Yaskawa INFORM job: SKRZYNIA_4040_180_STOPNI_10B_NEW.JBI

/JOB
//NAME SKRZYNIA_4040_180_STOPNI_10B_NEW
///FOLDERNAME 02-SKRZYNIE_JOBS
//POS
///NPOS 723,723,0,26,0,0
///TOOL 0
///POSTYPE PULSE
///PULSE
C00000=-21231,-51303,42314,2367,6591,-1439
C00001=-12854,-61498,-6635,149088,-29435,16513
C00002=84284,-61498,-6635,149088,14842,16513
C00003=84426,-61498,-62039,149088,14842,16513
C00004=84426,-61498,-83719,149088,14842,16513
C00005=40079,-25830,-61904,72398,37828,17494
C00006=40079,-25830,-61904,72398,37828,17494
C00007=38824,-23395,-60038,72349,38727,17731
C00008=41545,-22667,-59464,70826,37145,18191
C00009=40079,-25830,-61904,72398,37828,17494
C00010=40079,-23879,-31232,97616,36989,2612
C00011=40241,-22903,-30855,97033,36795,2952
C00012=39596,-21803,-29985,96678,37187,3182
C00013=41542,-21522,-29763,96797,35874,3054
C00014=40241,-22903,-30855,97033,36795,2952
C00015=44500,-22967,-34027,49689,40772,15208
C00016=44759,-21950,-33222,49364,40770,15399
C00017=43898,-20603,-32137,49608,41392,15289
C00018=45676,-20288,-31878,48567,40497,15854
C00019=44759,-21950,-33222,49364,40770,15399
C00020=50639,-31838,-53853,40430,42590,20636
C00021=47737,-42531,-47731,84740,46626,-3202
C00022=73324,-51450,-15857,136644,48513,-27329
C00023=28578,-31257,-33285,101874,54895,-3139
C00024=29101,-23166,-41439,93785,52323,3372
C00025=30342,-16402,-40775,90158,51109,6027
C00026=29555,-14242,-38855,90054,51607,6222
C00027=31304,-14182,-38798,89754,50458,6198
C00028=30342,-16402,-40775,90158,51109,6027
C00029=37840,-26567,-47806,97824,39338,5403
C00030=38314,-22656,-45541,96192,38787,6352
C00031=38740,-21749,-44817,95954,38481,6451
C00032=38106,-20505,-43805,95701,38856,6673
C00033=39920,-20274,-43616,95549,37666,6573
C00034=38740,-21749,-44817,95954,38481,6451
C00035=35154,-23288,-28184,89821,43405,2441
C00036=35403,-21021,-26397,89340,43215,2751
C00037=34678,-19569,-25213,89063,43699,2948
C00038=36545,-19419,-25091,89018,42427,2940
C00039=35403,-21021,-26397,89340,43215,2751
C00040=46673,-28267,-59493,36306,49500,22578
C00041=47298,-25083,-54483,36432,48421,22382
C00042=46134,-23276,-53085,36983,49197,22170
C00043=48093,-22778,-52692,35651,48513,22818
C00044=47298,-25083,-54483,36432,48421,22382
C00045=72417,-67880,-88171,46465,42262,31903
C00046=81480,-74508,-67932,111005,17511,3722
C00047=42492,-36415,-29790,92406,42740,11684
C00048=46673,-28267,-59493,36306,49500,22578
C00049=47298,-25083,-54483,36432,48421,22382
C00050=46134,-23276,-53085,36983,49197,22170
C00051=48093,-22778,-52692,35651,48513,22818
C00052=47298,-25083,-54483,36432,48421,22382
C00053=46673,-28267,-59493,36306,49500,22578
C00054=47298,-25083,-54483,36432,48421,22382
C00055=46134,-23276,-53085,36983,49197,22170
C00056=48093,-22778,-52692,35651,48513,22818
C00057=47309,-25052,-54460,36421,48423,22388
C00058=43000,-32780,-49011,53703,41088,15214
C00059=66148,-65994,-55487,105361,28212,-7739
C00060=66148,-65994,-55487,105361,28212,-7739
C00061=59848,-54778,-49507,133915,29212,-10807
C00062=45497,-38347,-41839,114412,32622,-465
C00063=46376,-32635,-46933,102993,29107,5780
C00064=46303,-28031,-46898,97061,28371,8976
C00065=45038,-26161,-45521,96183,29128,9541
C00066=46946,-25787,-45238,96120,27855,9431
C00067=46303,-28031,-46898,97061,28371,8976
C00068=45864,-17128,1685,129467,40696,-9274
C00069=46023,-15894,1830,128891,40053,-8896
C00070=45181,-14790,2774,128176,40341,-8535
C00071=46921,-14545,2986,129317,39465,-9073
C00072=45402,-17127,796,128656,40504,-8810
C00073=42828,-21985,-11573,106778,34538,-1929
C00074=43349,-21404,-11124,106831,34165,-1930
C00075=42250,-19876,-9917,105946,34757,-1485
C00076=44494,-19460,-9583,106781,33302,-1837
C00077=42797,-21858,-11474,106726,34550,-1903
C00078=42956,-14057,7354,88292,32197,-569
C00079=43438,-13569,7781,88275,31880,-510
C00080=42549,-12302,8904,87823,32462,-349
C00081=44721,-11883,9282,88161,31033,-316
C00082=42944,-14884,6642,88491,32210,-682
C00083=72417,-67880,-88171,46465,42262,31903
C00084=81480,-74508,-67932,111005,17511,3722
C00085=42492,-36415,-29790,92406,42740,11684
C00086=29699,-14901,-14062,86637,51249,15251
C00087=28921,-12904,-12269,86425,51786,15406
C00088=30978,-12767,-12144,86426,50380,15429
C00089=29506,-17416,-16239,86937,51377,15018
C00090=88410,-69609,-60867,139529,19008,-8209
C00091=62412,-62489,-12046,-12266,17816,34850
C00092=7585,-53665,33325,-3309,7810,4157
C00093=-681,-52632,38645,-5695,5489,-631
C00094=-17840,-61498,-6635,-149088,-29435,-16513
C00095=-84284,-61498,-6635,-149088,14842,-16513
C00096=-84426,-61498,-62039,-149088,14842,-16513
C00097=-84426,-61498,-83719,-149088,14842,-16513
C00098=-83351,-27062,-60322,-167360,37385,6517
C00099=-83351,-27062,-60322,-167360,37385,23281
C00100=-45097,-23850,-79932,-76262,26943,-22849
C00101=-48253,-15729,-73342,-71138,25693,-24842
C00102=-50302,-13076,-73239,-65836,25323,-27140
C00103=-49401,-11675,-71961,-66260,25816,-27133
C00104=-50608,-11574,-71867,-65226,25249,-27391
C00105=-49660,-13361,-73494,-66442,25615,-26975
C00106=-48242,-21102,-77802,-73044,25430,-23851
C00107=-42432,-29691,-46140,-101591,34194,-3953
C00108=-40467,-32259,-45349,-89481,35752,-6083
C00109=-35590,-22323,-38089,-87474,43148,-7978
C00110=-34853,-20780,-36847,-87247,43643,-8181
C00111=-37029,-20471,-36594,-86926,42180,-8224
C00112=-35503,-23333,-38886,-87700,43207,-7835
C00113=-41659,-25848,-37197,-61468,39541,-12344
C00114=-42019,-23363,-32043,-63110,38591,-11327
C00115=-41283,-22167,-31102,-63128,39154,-11341
C00116=-43189,-21868,-30866,-62281,38009,-11788
C00117=-40846,-25460,-35158,-62968,39555,-11455
C00118=-39561,-32409,-42051,-71473,38885,-9254
C00119=-88477,-67032,-53890,-125185,13082,17955
C00120=-90715,-66667,-50935,-152816,24533,28486
C00121=-30735,-26920,-32844,-95116,50209,-1071
C00122=-37180,-24683,-31930,-114741,47007,2943
C00123=-36407,-19634,-34656,-109847,45004,-453
C00124=-38352,-16604,-33863,-108521,43129,-1176
C00125=-37479,-14809,-32279,-108169,43576,-1482
C00126=-39395,-14487,-31992,-108361,42368,-1194
C00127=-37253,-18321,-35339,-108644,43916,-1187
C00128=-30948,-19486,-27368,-89515,49970,-2899
C00129=-32453,-17458,-25663,-89179,48933,-3088
C00130=-31896,-16151,-24534,-89028,49305,-3221
C00131=-33527,-16125,-24510,-88960,48196,-3202
C00132=-31291,-18911,-26892,-89421,49733,-2955
C00133=-32789,-14788,-10714,-75998,48642,-1904
C00134=-33953,-13481,-9550,-75758,47902,-2112
C00135=-33380,-12226,-8408,-75670,48319,-2157
C00136=-35020,-12164,-8351,-75529,47228,-2306
C00137=-33300,-14767,-10697,-75957,48300,-1949
C00138=-33300,-14767,-10697,-75957,48300,-1949
C00139=-33901,-13199,-7224,-76945,47663,-1266
C00140=-33178,-11617,-5779,-76815,48184,-1329
C00141=-35129,-11426,-5603,-76688,46886,-1497
C00142=-32900,-14718,-9841,-76444,48459,-1584
C00143=-74406,-60637,-53290,-78600,32734,-4861
C00144=-66351,-49775,-22313,-121187,42752,19491
C00145=-38126,-18978,-6321,-103556,42156,4232
C00146=-33300,-14767,-10697,-75957,48300,-1949
C00147=-33901,-13199,-7224,-76945,47663,-1266
C00148=-33178,-11617,-5779,-76815,48184,-1329
C00149=-35129,-11426,-5603,-76688,46886,-1497
C00150=-32900,-14718,-9841,-76444,48459,-1584
C00151=-33300,-14767,-10697,-75957,48300,-1949
C00152=-33901,-13199,-7224,-76945,47663,-1266
C00153=-33178,-11617,-5779,-76815,48184,-1329
C00154=-35129,-11426,-5603,-76688,46886,-1497
C00155=-33596,-13726,-8578,-76506,47971,-1566
C00156=-46324,-38325,-53351,-48650,39022,-16558
C00157=-84678,-53272,-42524,-56273,5220,-14251
C00158=-79949,-57830,-54545,-43165,18800,-25262
C00159=-85199,-63426,-59279,-35356,8253,-25340
C00160=-43240,-40066,-69296,-76804,34492,-13950
C00161=-32352,-24302,-62495,-76398,48702,-17646
C00162=-33867,-19497,-59989,-74208,48202,-18898
C00163=-33043,-17469,-58279,-74274,48770,-19034
C00164=-35172,-17180,-58031,-73305,47532,-19251
C00165=-33150,-20833,-61090,-74721,48572,-18687
C00166=-32525,-19963,-22291,-97454,48417,-2656
C00167=-34479,-17146,-19937,-97221,47013,-2812
C00168=-33716,-15515,-18525,-96928,47480,-3025
C00169=-35357,-15455,-18472,-97073,46375,-2908
C00170=-33341,-18474,-21063,-97306,47817,-2759
C00171=-32838,-10388,7981,-94473,48357,2926
C00172=-33747,-9461,8037,-94117,47673,2571
C00173=-33094,-8062,9377,-93861,48090,2458
C00174=-34952,-7927,9507,-94260,46861,2543
C00175=-33010,-10379,7174,-94037,48174,2591
C00176=-36099,-20774,-22249,-70758,44565,-7624
C00177=-37926,-16067,-12890,-73276,42575,-5996
C00178=-37323,-14944,-11908,-73188,43017,-6038
C00179=-39053,-14785,-11769,-72915,41882,-6255
C00180=-37847,-19214,-17221,-72670,42783,-6386
C00181=-74406,-60637,-53290,-78600,32734,-4861
C00182=-66351,-49775,-22313,-121187,42752,19491
C00183=-38126,-18978,-6321,-103556,42156,4232
C00184=-39485,-17529,-8330,-90200,39091,223
C00185=-38315,-15563,-6658,-89669,39866,-39
C00186=-40130,-15376,-6497,-89855,38637,-21
C00187=-40610,-23081,-12745,-91737,38407,1092
C00188=-82794,-45547,-18103,-153793,26453,27163
C00189=-46099,-67236,-11725,-98004,28606,19827
C00190=275,-40498,62911,330,272,-175
C00191=-21231,-51303,42314,2367,6591,-1439
C00192=-12854,-61498,-6635,149088,-29435,16513
C00193=84284,-61498,-6635,149088,14842,16513
C00194=84426,-61498,-62039,149088,14842,16513
C00195=84426,-61498,-83719,149088,14842,16513
C00196=40079,-25830,-61904,72398,37828,17494
C00197=43542,-21744,-53414,85694,32141,12908
C00198=43538,-20959,-59091,78847,32551,16732
C00199=40079,-23879,-31232,97616,36989,2612
C00200=41069,-22296,-36683,87871,35939,7163
C00201=41069,-20857,-27994,94343,36275,3375
C00202=40241,-22903,-30855,97033,36795,2952
C00203=44500,-22967,-34027,49689,40772,15208
C00204=37674,-14410,-29425,54908,51799,12689
C00205=37617,-13106,-20810,58248,49229,10178
C00206=44759,-21950,-33222,49364,40770,15399
C00207=50639,-31838,-53853,40430,42590,20636
C00208=47737,-42531,-47731,84740,46626,-3202
C00209=78714,-49092,-28755,133609,38199,-24420
C00210=28578,-31257,-33285,101874,54895,-3139
C00211=29101,-23166,-41439,93785,52323,3372
C00212=31163,-13872,-34138,92103,50752,4440
C00213=31163,-14064,-41434,88282,50498,7326
C00214=30342,-16402,-40775,90158,51109,6027
C00215=37840,-26567,-47806,97824,39338,5403
C00216=38314,-22656,-45541,96192,38787,6352
C00217=39658,-19881,-39017,99036,38353,4498
C00218=39658,-20227,-46296,93241,37598,7980
C00219=38740,-21749,-44817,95954,38481,6451
C00220=35154,-23288,-28184,89821,43405,2441
C00221=36302,-20456,-32356,81251,42995,6506
C00222=36302,-19046,-24537,85721,42698,3608
C00223=35403,-21021,-26397,89340,43215,2751
C00224=46673,-28267,-59493,36306,49500,22578
C00225=35383,-14910,-45807,52457,59655,19882
C00226=35383,-15025,-38926,54776,56903,17744
C00227=47298,-25083,-54483,36432,48421,22382
C00228=72417,-64226,-72669,53660,37323,27470
C00229=81480,-74508,-67932,111005,17511,3722
C00230=31559,-23192,-27729,97069,50041,14774
C00231=31559,-23192,-27729,97069,50041,14774
C00232=46673,-28267,-59493,36306,49500,22578
C00233=37754,-20085,-42350,56977,49558,11229
C00234=37583,-19171,-35264,59813,47966,9525
C00235=50836,-29533,-47785,41620,34114,14584
C00236=46673,-28267,-59493,36306,49500,22578
C00237=35383,-14910,-45807,52457,59655,19882
C00238=35383,-15025,-38926,54776,56903,17744
C00239=40792,-20879,-47843,46282,52305,19657
C00240=43000,-32780,-49011,53703,41088,15214
C00241=90538,-65158,-52413,145953,6697,-22013
C00242=90538,-65158,-52413,145953,6697,-22013
C00243=59848,-54778,-49507,133915,29212,-10807
C00244=45497,-38347,-41839,114412,32622,-465
C00245=46376,-32635,-46933,102993,29107,5780
C00246=38443,-20223,-37840,96971,39567,10287
C00247=38443,-20698,-44956,91660,38993,13539
C00248=46303,-28031,-46898,97061,28371,8976
C00249=45864,-17128,1685,129467,40696,-9274
C00250=38069,-7942,12691,120284,49952,-5070
C00251=38069,-11604,1369,116685,47266,-2469
C00252=45402,-17127,796,128656,40504,-8810
C00253=42828,-21985,-11573,106778,34538,-1929
C00254=33281,-15275,-13406,92642,47209,4970
C00255=33281,-12456,-2996,97026,47894,1870
C00256=42797,-21858,-11474,106726,34550,-1903
C00257=42956,-14057,7354,88292,32197,-569
C00258=35915,-8349,8335,81338,43542,2014
C00259=35915,-4149,20758,86814,43229,-1568
C00260=42944,-14884,6642,88491,32210,-682
C00261=72417,-64226,-72669,53660,37323,27470
C00262=81480,-74508,-67932,111005,17511,3722
C00263=31559,-23192,-27729,97069,50041,14774
C00264=31559,-23192,-27729,97069,50041,14774
C00265=34921,-13948,-26935,108215,46513,15013
C00266=34921,-14719,-34056,104413,45059,17611
C00267=30729,-14807,-22031,91030,50318,16982
C00268=30729,-14807,-22031,91030,50318,16982
C00269=30729,-13019,-13516,94566,50766,14318
C00270=88410,-69609,-60867,139529,19008,-8209
C00271=62412,-62489,-12046,-12266,17816,34850
C00272=-245,-52407,39795,-2053,6376,-227
C00273=-681,-52632,38645,-5695,5489,-631
C00274=-17840,-61498,-6635,-149088,-29435,-16513
C00275=-84284,-61498,-6635,-149088,14842,-16513
C00276=-84426,-61498,-62039,-149088,14842,-16513
C00277=-84426,-61498,-83719,-149088,14842,-16513
C00278=-83351,-27062,-60322,-167360,37385,6517
C00279=-83351,-27062,-60322,-167360,37385,23281
C00280=-45097,-23850,-79932,-76262,26943,-22849
C00281=-48253,-15729,-73342,-71138,25693,-24842
C00282=-42869,-6204,-67496,-75794,33821,-25861
C00283=-42869,-3205,-70686,-69723,34977,-29338
C00284=-49660,-13361,-73494,-66442,25615,-26975
C00285=-48242,-21102,-77802,-73044,25430,-23851
C00286=-42432,-29691,-46140,-101591,34194,-3953
C00287=-40467,-32259,-45349,-89481,35752,-6083
C00288=-32032,-15700,-34761,-86363,49905,-9645
C00289=-32032,-14866,-27372,-89947,49973,-6979
C00290=-35503,-23333,-38886,-87700,43207,-7835
C00291=-41659,-25848,-37197,-61468,39541,-12344
C00292=-32550,-13183,-23016,-68651,53358,-8526
C00293=-34023,-12481,-22084,-63241,53452,-9524
C00294=-40846,-25460,-35158,-62968,39555,-11455
C00295=-39561,-32409,-42051,-71473,38885,-9254
C00296=-88477,-67032,-53890,-125185,13082,17955
C00297=-90715,-66667,-50935,-152816,24533,28486
C00298=-30735,-26920,-32844,-95116,50209,-1071
C00299=-37180,-24683,-31930,-114741,47007,2943
C00300=-36407,-19634,-34656,-109847,45004,-453
C00301=-39264,-14095,-28560,-110319,43249,69
C00302=-39254,-14742,-35710,-105973,41627,-2729
C00303=-37253,-18321,-35339,-108644,43916,-1187
C00304=-30948,-19486,-27368,-89515,49970,-2899
C00305=-33188,-17217,-33290,-80523,49125,-7157
C00306=-33231,-16133,-25752,-84153,48705,-4513
C00307=-31291,-18911,-26892,-89421,49733,-2955
C00308=-32789,-14788,-10714,-75998,48642,-1904
C00309=-32456,-10000,-8763,-74569,51725,-2878
C00310=-32456,-7502,814,-78111,50801,-165
C00311=-33300,-14767,-10697,-75957,48300,-1949
C00312=-33300,-14767,-10697,-75957,48300,-1949
C00313=-31039,-7597,-4415,-75714,54029,-1891
C00314=-31745,-5891,1281,-74609,53027,-1007
C00315=-32900,-14718,-9841,-76444,48459,-1584
C00316=-73757,-59015,-49060,-81128,30370,-3444
C00317=-66351,-49775,-22313,-115582,40632,19491
C00318=-39230,-13378,9505,-118180,46878,7841
C00319=-33300,-14767,-10697,-75957,48300,-1949
C00320=-31039,-7597,-4415,-75714,54029,-1891
C00321=-31745,-5891,1281,-74609,53027,-1007
C00322=-32900,-14718,-9841,-76444,48459,-1584
C00323=-33300,-14767,-10697,-75957,48300,-1949
C00324=-31039,-7597,-4415,-75714,54029,-1891
C00325=-31745,-5891,1281,-74609,53027,-1007
C00326=-31800,-10328,-6603,-75899,51910,-1826
C00327=-46324,-38325,-53351,-48650,39022,-16558
C00328=-84678,-53272,-42524,-56273,5220,-14251
C00329=-79949,-57830,-54545,-43165,18800,-25262
C00330=-85199,-63426,-59279,-35356,8253,-25340
C00331=-43240,-40066,-69296,-76804,34492,-13950
C00332=-32352,-24302,-62495,-76398,48702,-17646
C00333=-34311,-15084,-43386,-89458,46770,-12174
C00334=-34303,-14562,-49859,-85086,46777,-15220
C00335=-33150,-20833,-61090,-74721,48572,-18687
C00336=-32525,-19963,-22291,-97454,48417,-2656
C00337=-35706,-13608,-12356,-102024,46946,-662
C00338=-35706,-15621,-21438,-97808,45877,-3577
C00339=-33341,-18474,-21063,-97306,47817,-2759
C00340=-32838,-10388,7981,-94473,48357,2926
C00341=-33093,-7396,5806,-90907,49596,566
C00342=-33114,-3922,16616,-94789,50065,3444
C00343=-33010,-10379,7174,-94037,48174,2591
C00344=-36099,-20774,-22249,-70758,44565,-7624
C00345=-34715,-11750,-12273,-72011,49148,-6727
C00346=-34715,-9605,-3694,-75523,48112,-4187
C00347=-37847,-19214,-17221,-72670,42783,-6386
C00348=-73757,-59015,-49060,-81128,30370,-3444
C00349=-66351,-49775,-22313,-115582,40632,19491
C00350=-39230,-13378,9505,-118180,46878,7841
C00351=-45382,-7236,12023,-133378,48537,9962
C00352=-45404,-10871,608,-130166,44845,7725
C00353=-39289,-13633,5656,-114159,44810,6160
C00354=-38323,-13232,3563,-106275,42852,3854
C00355=-39624,-12309,2722,-105485,41613,3229
C00356=-39624,-8328,14658,-110578,43519,6514
C00357=-36264,-16485,7382,-110054,45980,6615
C00358=-44249,-32643,-4456,-118298,43922,12613
C00359=-31781,-48654,10305,-108801,40875,18482
C00360=275,-40498,62911,330,272,-175
C00361=-21231,-51303,42314,2367,6591,-1439
C00362=-12854,-61498,-6635,149088,-29435,16513
C00363=1243,-64916,-20173,127712,-3737,19309
C00364=25728,-72945,-47671,86292,40512,26238
C00365=76664,-93599,-96338,114349,24908,7990
C00366=72545,-76403,-90681,98079,12187,16258
C00367=68435,-42241,-79282,43384,21203,43145
C00368=65057,-16377,-54230,51764,24572,24912
C00369=65057,-16377,-54230,51764,24572,24912
C00370=63338,-14509,-52578,53100,25585,24479
C00371=65493,-13068,-51269,50530,24633,25485
C00372=65057,-16377,-54230,51764,24572,24912
C00373=65057,-15356,-24189,99795,20011,765
C00374=64877,-14372,-23690,98704,20045,1316
C00375=64002,-13489,-22890,98156,20604,1621
C00376=65592,-12702,-22173,98357,19527,1466
C00377=64877,-14372,-23690,98704,20045,1316
C00378=68341,-13254,-25781,29903,31229,25524
C00379=68283,-12212,-24821,29865,31356,25548
C00380=67188,-11145,-23825,30867,31841,25051
C00381=68624,-10377,-23095,29361,31405,25809
C00382=68283,-12212,-24821,29865,31356,25548
C00383=67373,-28813,-51747,26561,36937,27500
C00384=65665,-56911,-59086,75825,31170,1181
C00385=86238,-56758,-47218,93606,16664,-7096
C00386=86238,-56758,-47218,93606,16664,-7096
C00387=58162,-25487,-29222,106212,35121,-6052
C00388=54729,-17550,-36821,90686,35172,3055
C00389=53879,-10723,-35593,84994,35691,6442
C00390=52628,-8898,-33837,85063,36512,6546
C00391=54193,-8333,-33282,84633,35489,6620
C00392=53879,-10723,-35593,84994,35691,6442
C00393=63265,-18185,-41125,95483,22448,4389
C00394=62561,-14368,-38517,92984,22773,5727
C00395=62689,-13396,-37636,92694,22678,5861
C00396=61812,-12400,-36718,92465,23238,6064
C00397=63331,-11679,-36046,92201,22238,6052
C00398=62689,-13396,-37636,92694,22678,5861
C00399=60836,-16142,-22303,87853,25853,3109
C00400=60346,-13901,-20318,87240,26185,3441
C00401=59279,-12702,-19226,86999,26911,3593
C00402=60868,-12050,-18626,86765,25831,3679
C00403=60346,-13901,-20318,87240,26185,3441
C00404=71174,-16943,-50501,16787,44328,31924
C00405=70846,-13961,-45205,17496,43056,31510
C00406=69412,-12602,-43961,18675,43507,30969
C00407=70949,-11616,-43043,17320,43301,31610
C00408=70846,-13961,-45205,17496,43056,31510
C00409=75423,-38775,-29488,68062,11357,11878
C00410=83800,-53438,-37305,103753,25026,-1265
C00411=73693,-43023,-29306,101200,31062,8332
C00412=71174,-16943,-50501,16787,44328,31924
C00413=70846,-13961,-45205,17496,43056,31510
C00414=69412,-12602,-43961,18675,43507,30969
C00415=70949,-11616,-43043,17320,43301,31610
C00416=70846,-13961,-45205,17496,43056,31510
C00417=71174,-16943,-50501,16787,44328,31924
C00418=70846,-13961,-45205,17496,43056,31510
C00419=69412,-12602,-43961,18675,43507,30969
C00420=70949,-11616,-43043,17320,43301,31610
C00421=70341,-14112,-45346,17938,43139,31306
C00422=66765,-25643,-43957,33958,30926,25005
C00423=89904,-51519,-74342,14421,36812,44678
C00424=59533,-60921,-66479,83565,41795,11392
C00425=74572,-27669,-34920,136415,14797,-11887
C00426=72479,-21736,-38943,108586,11547,1590
C00427=70901,-17325,-38411,94105,11830,8638
C00428=69318,-15905,-37172,92885,12849,9347
C00429=70820,-15051,-36412,92531,11846,9399
C00430=70901,-17325,-38411,94105,11830,8638
C00431=70927,-7523,10343,151197,29871,-19432
C00432=70517,-6236,10737,150221,29352,-18933
C00433=69462,-5331,11645,148944,29606,-18324
C00434=70849,-4645,12343,150548,29173,-19084
C00435=70402,-7634,9356,150158,29478,-18907
C00436=68660,-13051,-4106,122816,18275,-8999
C00437=68895,-12351,-3471,122899,18094,-9031
C00438=67458,-11121,-2337,120787,18802,-8043
C00439=69212,-10147,-1425,122703,17774,-8922
C00440=68590,-12934,-4000,122687,18305,-8939
C00441=67960,-5141,15741,92957,15720,-628
C00442=68207,-4523,16370,92944,15555,-601
C00443=67051,-3465,17460,92338,16311,-404
C00444=68762,-2475,18496,92897,15183,-531
C00445=68227,-5981,14898,93242,15553,-745
C00446=75423,-38775,-29488,68062,11357,11878
C00447=83800,-53438,-37305,103753,25026,-1265
C00448=73693,-43023,-29306,101200,31062,8332
C00449=57182,-8361,13896,122065,42938,1264
C00450=54175,-4244,10116,111777,38351,4895
C00451=53015,-2664,11762,111180,39035,5172
C00452=54334,-2350,12093,111780,38228,4906
C00453=54175,-4244,10116,111777,38351,4895
C00454=89016,-59505,-36896,143842,20811,-11822
C00455=0,-52280,40443,0,6876,0
C00456=-681,-52632,38645,-5695,5489,-631
C00457=-17840,-61498,-6635,-149088,-29435,-16513
C00458=-84284,-61498,-6635,-149088,14842,-16513
C00459=-57949,-92832,-68327,-119114,39180,-13331
C00460=-51160,-78996,-68705,-103851,38676,-21739
C00461=-70129,-12201,-70194,-45988,15849,-32683
C00462=-70861,-4247,-62448,-43170,16032,-33903
C00463=-72229,-1292,-61598,-37253,16795,-36501
C00464=-71164,-286,-60510,-39045,17142,-35862
C00465=-72168,114,-60071,-37345,16819,-36474
C00466=-71747,-1710,-62044,-38091,16943,-36199
C00467=-72086,-8949,-67137,-41785,15362,-34318
C00468=-68226,-19972,-38714,-103620,16923,-1218
C00469=-67549,-22986,-38612,-80975,17520,-9124
C00470=-60286,-14955,-31870,-81576,26630,-9634
C00471=-59206,-13694,-30736,-81541,27366,-9725
C00472=-61026,-12796,-29913,-80837,26167,-9971
C00473=-60502,-15936,-32740,-81790,26471,-9505
C00474=-66711,-16726,-29834,-42060,26790,-21996
C00475=-66477,-14329,-24475,-44917,25565,-20507
C00476=-65503,-13376,-23611,-45716,26132,-20127
C00477=-67048,-12587,-22889,-44009,25442,-20959
C00478=-66009,-16611,-27996,-44380,26285,-20808
C00479=-67084,-23473,-35621,-52822,22843,-18344
C00480=-54372,-63877,-56403,-90862,27079,1323
C00481=-55608,-75012,-34654,-126966,55573,20814
C00482=-55608,-75012,-34654,-126966,55573,20814
C00483=-58069,-20780,-28125,-95622,31565,-134
C00484=-62818,-16895,-25617,-123146,31403,8811
C00485=-60301,-12189,-28106,-114654,29999,4030
C00486=-61167,-8731,-26593,-112607,28768,2985
C00487=-59960,-7252,-25135,-111997,29446,2563
C00488=-61574,-6413,-24296,-112502,28453,2957
C00489=-60636,-10677,-28466,-112685,29164,2987
C00490=-55814,-13636,-22293,-87541,33030,-3263
C00491=-56566,-11270,-20110,-87077,32519,-3496
C00492=-55709,-10167,-19066,-86969,33101,-3589
C00493=-57154,-9687,-18605,-86794,32120,-3632
C00494=-55949,-12989,-21706,-87412,32939,-3330
C00495=-57109,-8613,-4995,-71756,32687,-5152
C00496=-57764,-7017,-3429,-71410,32292,-5358
C00497=-56909,-5946,-2356,-71529,32873,-5273
C00498=-58347,-5433,-1836,-71115,31941,-5534
C00499=-57555,-8453,-4841,-71622,32398,-5235
C00500=-57555,-8453,-4841,-71622,32398,-5235
C00501=-57844,-6749,-1100,-73475,31868,-4209
C00502=-56760,-5394,262,-73573,32605,-4123
C00503=-58439,-4668,1002,-73167,31507,-4396
C00504=-57269,-8513,-4090,-72514,32435,-4729
C00505=-69972,-70945,-58827,-87515,35615,-17
C00506=-69972,-70945,-58827,-87515,35615,-17
C00507=-64053,-11295,342,-114563,25508,8776
C00508=-57555,-8453,-4841,-71622,32398,-5235
C00509=-57844,-6749,-1100,-73475,31868,-4209
C00510=-56760,-5394,262,-73573,32605,-4123
C00511=-58439,-4668,1002,-73167,31507,-4396
C00512=-57269,-8513,-4090,-72514,32435,-4729
C00513=-57555,-8453,-4841,-71622,32398,-5235
C00514=-57844,-6749,-1100,-73475,31868,-4209
C00515=-56760,-5394,262,-73573,32605,-4123
C00516=-58439,-4668,1002,-73167,31507,-4396
C00517=-57340,-8164,-3656,-72551,32379,-4710
C00518=-74194,-26905,-45748,-21164,30431,-30370
C00519=-93036,-61583,-83098,-4972,39040,-38907
C00520=-93036,-61583,-83098,-4972,39040,-38907
C00521=-71878,-28414,-61729,-48672,19032,-25171
C00522=-58025,-17185,-56692,-61796,34178,-22014
C00523=-58138,-12270,-53641,-59720,34855,-23185
C00524=-56898,-10637,-52111,-60384,35596,-23031
C00525=-58712,-9745,-51261,-58987,34681,-23500
C00526=-57851,-13714,-54968,-60141,34926,-22995
C00527=-57767,-13689,-16896,-100181,31334,-836
C00528=-58645,-10437,-13885,-99794,30663,-1040
C00529=-57513,-9065,-12573,-99347,31388,-1300
C00530=-58947,-8556,-12078,-99591,30423,-1148
C00531=-58031,-12031,-15383,-99926,31110,-974
C00532=-57646,-4162,14084,-101426,32077,4804
C00533=-58050,-2999,14481,-100683,31666,4357
C00534=-57067,-1784,15765,-100255,32298,4198
C00535=-58672,-1130,16464,-100866,31256,4407
C00536=-57676,-4116,13320,-100600,31921,4338
C00537=-61201,-13510,-16039,-60848,29053,-13371
C00538=-61885,-8475,-5914,-65722,27292,-10768
C00539=-61040,-7537,-4993,-65975,27855,-10622
C00540=-62506,-6917,-4380,-65230,26947,-11038
C00541=-62587,-11561,-10517,-63923,27184,-11731
C00542=-69972,-70945,-58827,-87515,35615,-17
C00543=-69972,-70945,-58827,-87515,35615,-17
C00544=-64053,-11295,342,-114563,25508,8776
C00545=-64305,-9514,-1154,-92513,22236,350
C00546=-62690,-7882,422,-91839,23314,70
C00547=-64201,-7220,1072,-92034,22288,112
C00548=-67149,-14673,-5883,-94845,20391,1413
C00549=-66017,-67071,-29713,-134523,32873,22112
C00550=-46099,-67236,-11725,-98004,28606,19827
C00551=275,-40498,62911,330,272,-175
C00552=-21231,-51303,42314,2367,6591,-1439
C00553=-12854,-61498,-6635,149088,-29435,16513
C00554=84284,-61498,-6635,149088,14842,16513
C00555=84426,-61498,-62039,149088,14842,16513
C00556=84426,-61498,-83719,149088,14842,16513
C00557=65057,-16377,-54230,51764,24572,24912
C00558=84197,-12836,-45810,-45141,8815,68584
C00559=84197,-12041,-51210,-30828,12194,61758
C00560=65057,-15356,-24189,99795,20011,765
C00561=74080,-15423,-30907,69143,7686,14038
C00562=74080,-14352,-23480,100923,7503,-991
C00563=64877,-14372,-23690,98704,20045,1316
C00564=68341,-13254,-25781,29903,31229,25524
C00565=74439,-11496,-26749,13621,29642,33649
C00566=74439,-10401,-19085,15788,25340,32499
C00567=68283,-12212,-24821,29865,31356,25548
C00568=75452,-19560,-44582,17787,36745,31835
C00569=68183,-44834,-62310,40554,34116,19994
C00570=94103,-63119,-69903,16230,17694,31762
C00571=91219,-55958,-51219,93435,14423,-1742
C00572=58162,-25487,-29222,106212,35121,-6052
C00573=54729,-17550,-36821,90686,35172,3055
C00574=70769,-15160,-35297,83470,11760,4000
C00575=70769,-15377,-40609,67973,12489,11436
C00576=53879,-10723,-35593,84994,35691,6442
C00577=63265,-18185,-41125,95483,22448,4389
C00578=62561,-14368,-38517,92984,22773,5727
C00579=77715,-13962,-33882,144680,4496,-21400
C00580=77806,-14046,-41277,60589,2532,18064
C00581=62689,-13396,-37636,92694,22678,5861
C00582=60836,-16142,-22303,87853,25853,3109
C00583=74678,-16514,-29029,42946,9451,23276
C00584=74678,-15315,-21920,65026,7151,12815
C00585=60346,-13901,-20318,87240,26185,3441
C00586=71174,-16943,-50501,16787,44328,31924
C00587=80494,-13102,-44599,-1731,38384,44653
C00588=80494,-13295,-38861,-1907,34285,44756
C00589=70846,-13961,-45205,17496,43056,31510
C00590=83595,-66668,-34414,154325,14846,-28455
C00591=83595,-66668,-34414,154325,14846,-28455
C00592=69137,-30288,-25983,94330,24536,11676
C00593=71174,-16943,-50501,16787,44328,31924
C00594=80494,-13102,-44599,-1731,38384,44653
C00595=80494,-13295,-38861,-1907,34285,44756
C00596=70846,-13961,-45205,17496,43056,31510
C00597=71056,-15939,-48723,17027,43904,31784
C00598=80494,-13102,-44599,-1731,38384,44653
C00599=80494,-13295,-38861,-1907,34285,44756
C00600=73484,-14077,-43720,13005,40199,34803
C00601=69645,-22678,-41665,30358,30421,26767
C00602=81017,-78801,-66317,80675,7786,2447
C00603=81017,-78801,-66317,80675,7786,2447
C00604=74572,-27669,-34920,136415,14797,-11887
C00605=72479,-21736,-38943,108586,11547,1590
C00606=76162,-15538,-34076,119407,5153,-4143
C00607=76225,-15803,-40874,66675,4586,20654
C00608=70901,-17325,-38411,94105,11830,8638
C00609=70927,-7523,10343,151197,29871,-19432
C00610=75273,-951,23395,164730,33684,-27271
C00611=75257,-4812,11918,163197,28775,-26429
C00612=70402,-7634,9356,150158,29478,-18907
C00613=68660,-13051,-4106,122816,18275,-8999
C00614=75422,-13779,-12311,124767,7049,-10125
C00615=75402,-11409,-3274,143452,10422,-18986
C00616=68590,-12934,-4000,122687,18305,-8939
C00617=67960,-5141,15741,92957,15720,-628
C00618=77005,-5383,11265,73049,3770,10304
C00619=77005,-1367,23224,135174,5603,-18901
C00620=68227,-5981,14898,93242,15553,-745
C00621=83595,-66668,-34414,154325,14846,-28455
C00622=83595,-66668,-34414,154325,14846,-28455
C00623=69137,-30288,-25983,94330,24536,11676
C00624=69694,-21959,-24250,77622,17543,9395
C00625=72869,1541,21011,161481,40400,-32944
C00626=75019,3768,21884,166311,43242,-33805
C00627=75946,3919,31956,167866,49928,-34763
C00628=66712,-14281,-1549,117281,20128,-19574
C00629=72038,-15960,-22039,53337,12147,14456
C00630=72038,-13517,-11162,79650,10019,1887
C00631=70769,-47931,-32777,112213,25945,2479
C00632=17178,-50520,12136,39169,20391,2344
C00633=-681,-52632,38645,-5695,5489,-631
C00634=-17840,-61498,-6635,-149088,-29435,-16513
C00635=-84284,-61498,-6635,-149088,14842,-16513
C00636=-84426,-61498,-62039,-149088,14842,-16513
C00637=-84426,-61498,-83719,-149088,14842,-16513
C00638=-83351,-27062,-60322,-167360,37385,6517
C00639=-83351,-27062,-60322,-167360,37385,23281
C00640=-70129,-12201,-70194,-45988,15849,-32683
C00641=-70861,-4247,-62448,-43170,16032,-33903
C00642=-76882,43,-60950,-14294,14755,-45201
C00643=-76882,3984,-64926,-10429,20329,-47102
C00644=-71747,-1710,-62044,-38091,16943,-36199
C00645=-72086,-8949,-67137,-41785,15362,-34318
C00646=-68226,-19972,-38714,-103620,16923,-1218
C00647=-67549,-22986,-38612,-80975,17520,-9124
C00648=-69143,-15166,-34287,-68804,15212,-14794
C00649=-69143,-14592,-28782,-80821,14459,-8960
C00650=-60502,-15936,-32740,-81790,26471,-9505
C00651=-66711,-16726,-29834,-42060,26790,-21996
C00652=-75652,-13136,-22972,-17539,18443,-33643
C00653=-76393,-11602,-18975,-13556,19574,-34543
C00654=-66009,-16611,-27996,-44380,26285,-20808
C00655=-61601,-28306,-39228,-59626,25389,-15050
C00656=-72315,-63222,-70224,-69600,33305,-10426
C00657=-72315,-63222,-70224,-69600,33305,-10426
C00658=-58069,-20780,-28125,-95622,31565,-134
C00659=-62818,-16895,-25617,-123146,31403,8811
C00660=-60301,-12189,-28106,-114654,29999,4030
C00661=-75089,-9933,-24682,-148597,14783,22922
C00662=-75089,-10642,-34451,-132584,9653,15243
C00663=-60636,-10677,-28466,-112685,29164,2987
C00664=-55814,-13636,-22293,-87541,33030,-3263
C00665=-73301,-16058,-32281,-44459,12702,-22095
C00666=-73339,-15052,-25249,-60236,10249,-14543
C00667=-55949,-12989,-21706,-87412,32939,-3330
C00668=-57109,-8613,-4995,-71756,32687,-5152
C00669=-71674,-10355,-9102,-48278,15013,-17468
C00670=-71670,-8088,-356,-62615,12652,-10541
C00671=-57555,-8453,-4841,-71622,32398,-5235
C00672=-57555,-8453,-4841,-71622,32398,-5235
C00673=-73349,-10209,-7254,-46090,12597,-18565
C00674=-73349,-7867,1452,-63091,10217,-10432
C00675=-57269,-8513,-4090,-72514,32435,-4729
C00676=-68334,-63389,-52515,-83837,33201,-1739
C00677=-68334,-63389,-52515,-83837,33201,-1739
C00678=-64053,-11295,342,-114563,25508,8776
C00679=-57555,-8453,-4841,-71622,32398,-5235
C00680=-73349,-10209,-7254,-46090,12597,-18565
C00681=-73349,-7867,1452,-63091,10217,-10432
C00682=-57269,-8513,-4090,-72514,32435,-4729
C00683=-57555,-8453,-4841,-71622,32398,-5235
C00684=-73349,-10209,-7254,-46090,12597,-18565
C00685=-70611,-8579,-7842,-39945,19879,-25243
C00686=-60697,-9016,-5571,-67071,28440,-8703
C00687=-74194,-26905,-45748,-21164,30431,-30370
C00688=-76007,-77202,-67157,-59280,11041,-11579
C00689=-76006,-77203,-67157,-59281,11043,-11581
C00690=-53398,-42726,-55849,-45492,34374,-18069
C00691=-71878,-28414,-61729,-48672,19032,-25171
C00692=-58025,-17185,-56692,-61796,34178,-22014
C00693=-77553,-14661,-43008,-35465,5780,-31120
C00694=-77553,-14004,-50514,-17997,10868,-39389
C00695=-57851,-13714,-54968,-60141,34926,-22995
C00696=-57767,-13689,-16896,-100181,31334,-836
C00697=-74769,-11126,-10073,-142523,13426,19686
C00698=-74753,-12848,-17783,-130765,10301,14051
C00699=-58031,-12031,-15383,-99926,31110,-974
C00700=-57646,-4162,14084,-101426,32077,4804
C00701=-72179,-7124,6017,-115427,12582,9833
C00702=-72179,-4103,15503,-129018,15105,16401
C00703=-57676,-4116,13320,-100600,31921,4338
C00704=-61201,-13510,-16039,-60848,29053,-13371
C00705=-74136,-10643,-11909,-32993,14820,-27251
C00706=-74162,-8377,-2780,-45377,11297,-21290
C00707=-62587,-11561,-10517,-63923,27184,-11731
C00708=-68334,-63389,-52515,-83837,33201,-1739
C00709=-68334,-63389,-52515,-83837,33201,-1739
C00710=-64053,-11295,342,-114563,25508,8776
C00711=-64053,-11295,342,-114563,25508,8776
C00712=-74239,7065,32887,-163372,44700,35065
C00713=-74142,3045,20239,-161993,39159,34198
C00714=-75119,4045,29308,-164063,44402,35406
C00715=-79833,-9558,5437,-165750,9898,43323
C00716=-75231,-7555,5870,-137998,10766,30530
C00717=-75231,-3987,16941,-149127,14978,35883
C00718=-77761,-13214,8113,-156332,15145,39163
C00719=-65551,-48104,-28924,-114827,24376,11665
C00720=-51220,-46814,3045,-130057,64886,23876
C00721=-46099,-67236,-11725,-98004,28606,19827
C00722=275,-40498,62911,330,272,-175
BC00000=467225
BC00001=513669
BC00002=494109
BC00003=467540
BC00004=467540
BC00005=478876
BC00006=478876
BC00007=478876
BC00008=478876
BC00009=478876
BC00010=478876
BC00011=478876
BC00012=478876
BC00013=478876
BC00014=478876
BC00015=478876
BC00016=478876
BC00017=478876
BC00018=478876
BC00019=478876
BC00020=478876
BC00021=481980
BC00022=563952
BC00023=606256
BC00024=606256
BC00025=606252
BC00026=606252
BC00027=606252
BC00028=606252
BC00029=654662
BC00030=654618
BC00031=654618
BC00032=654618
BC00033=654618
BC00034=654618
BC00035=654618
BC00036=654618
BC00037=654618
BC00038=654618
BC00039=654618
BC00040=686402
BC00041=686402
BC00042=686350
BC00043=686350
BC00044=686402
BC00045=680656
BC00046=761251
BC00047=725268
BC00048=747845
BC00049=747845
BC00050=747793
BC00051=747793
BC00052=747845
BC00053=778567
BC00054=778567
BC00055=778515
BC00056=778515
BC00057=753737
BC00058=652574
BC00059=648164
BC00060=761837
BC00061=767278
BC00062=762734
BC00063=769582
BC00064=784046
BC00065=784046
BC00066=784046
BC00067=784046
BC00068=784046
BC00069=784046
BC00070=784046
BC00071=784046
BC00072=784046
BC00073=821134
BC00074=821134
BC00075=821134
BC00076=821134
BC00077=821134
BC00078=821134
BC00079=821134
BC00080=821134
BC00081=821134
BC00082=821134
BC00083=757461
BC00084=838056
BC00085=802073
BC00086=809753
BC00087=809753
BC00088=809753
BC00089=809753
BC00090=838056
BC00091=718134
BC00092=692175
BC00093=518986
BC00094=509920
BC00095=467540
BC00096=467540
BC00097=467540
BC00098=521167
BC00099=520352
BC00100=535759
BC00101=535759
BC00102=535757
BC00103=535757
BC00104=535757
BC00105=535757
BC00106=535757
BC00107=485653
BC00108=485653
BC00109=485653
BC00110=485653
BC00111=485653
BC00112=485653
BC00113=485653
BC00114=485653
BC00115=485653
BC00116=485653
BC00117=485653
BC00118=485653
BC00119=485653
BC00120=615112
BC00121=615112
BC00122=615112
BC00123=615112
BC00124=615112
BC00125=615112
BC00126=615112
BC00127=615112
BC00128=615112
BC00129=615112
BC00130=615112
BC00131=615112
BC00132=615112
BC00133=615112
BC00134=615112
BC00135=615112
BC00136=615112
BC00137=615112
BC00138=658076
BC00139=658076
BC00140=658076
BC00141=658076
BC00142=658076
BC00143=658078
BC00144=722785
BC00145=722785
BC00146=719519
BC00147=719519
BC00148=719519
BC00149=719519
BC00150=719519
BC00151=750241
BC00152=750241
BC00153=750241
BC00154=750241
BC00155=723518
BC00156=655680
BC00157=643721
BC00158=643721
BC00159=793396
BC00160=799070
BC00161=799070
BC00162=799070
BC00163=799070
BC00164=799070
BC00165=799070
BC00166=799070
BC00167=799070
BC00168=799070
BC00169=799070
BC00170=799070
BC00171=799070
BC00172=799070
BC00173=799070
BC00174=799070
BC00175=799070
BC00176=845667
BC00177=845667
BC00178=845667
BC00179=845667
BC00180=845667
BC00181=734883
BC00182=799590
BC00183=799590
BC00184=799590
BC00185=799590
BC00186=799590
BC00187=799590
BC00188=799590
BC00189=764911
BC00190=508839
BC00191=467225
BC00192=513669
BC00193=494109
BC00194=467540
BC00195=467540
BC00196=478876
BC00197=478876
BC00198=478876
BC00199=478876
BC00200=478876
BC00201=478876
BC00202=478876
BC00203=478876
BC00204=478876
BC00205=478876
BC00206=478876
BC00207=478876
BC00208=481980
BC00209=584323
BC00210=606256
BC00211=606256
BC00212=606252
BC00213=606252
BC00214=606252
BC00215=654662
BC00216=654618
BC00217=654618
BC00218=654618
BC00219=654618
BC00220=654618
BC00221=654618
BC00222=654618
BC00223=654618
BC00224=686402
BC00225=686402
BC00226=686402
BC00227=686402
BC00228=680656
BC00229=759706
BC00230=759706
BC00231=759706
BC00232=747845
BC00233=747845
BC00234=747845
BC00235=747845
BC00236=778568
BC00237=778568
BC00238=778568
BC00239=758331
BC00240=652574
BC00241=641414
BC00242=715810
BC00243=784046
BC00244=784046
BC00245=784046
BC00246=784046
BC00247=784046
BC00248=784046
BC00249=784046
BC00250=784043
BC00251=784043
BC00252=784046
BC00253=821134
BC00254=821134
BC00255=821134
BC00256=821134
BC00257=821134
BC00258=821134
BC00259=821134
BC00260=821134
BC00261=757461
BC00262=836511
BC00263=836511
BC00264=836511
BC00265=836511
BC00266=836511
BC00267=836511
BC00268=836511
BC00269=836511
BC00270=841401
BC00271=717529
BC00272=644098
BC00273=472903
BC00274=509920
BC00275=467540
BC00276=467540
BC00277=467540
BC00278=521167
BC00279=520352
BC00280=535759
BC00281=535759
BC00282=535757
BC00283=535757
BC00284=535757
BC00285=535757
BC00286=485653
BC00287=485653
BC00288=485653
BC00289=485653
BC00290=485653
BC00291=485653
BC00292=485653
BC00293=485653
BC00294=485653
BC00295=485653
BC00296=485653
BC00297=615112
BC00298=615112
BC00299=615112
BC00300=615112
BC00301=615112
BC00302=615112
BC00303=615112
BC00304=615112
BC00305=615112
BC00306=615112
BC00307=615112
BC00308=615112
BC00309=615112
BC00310=615112
BC00311=615112
BC00312=658076
BC00313=658076
BC00314=658076
BC00315=658076
BC00316=641496
BC00317=715104
BC00318=725536
BC00319=719519
BC00320=719519
BC00321=719519
BC00322=719519
BC00323=750242
BC00324=750242
BC00325=750242
BC00326=735844
BC00327=655680
BC00328=643721
BC00329=643721
BC00330=793396
BC00331=799070
BC00332=799070
BC00333=799070
BC00334=799070
BC00335=799070
BC00336=799070
BC00337=799070
BC00338=799070
BC00339=799070
BC00340=799070
BC00341=799070
BC00342=799070
BC00343=799070
BC00344=845667
BC00345=845667
BC00346=845667
BC00347=845667
BC00348=718301
BC00349=791909
BC00350=802341
BC00351=802341
BC00352=802341
BC00353=802341
BC00354=811717
BC00355=811717
BC00356=811717
BC00357=811717
BC00358=800617
BC00359=741121
BC00360=639407
BC00361=467225
BC00362=406578
BC00363=397670
BC00364=437429
BC00365=535309
BC00366=478364
BC00367=478364
BC00368=478876
BC00369=478876
BC00370=478876
BC00371=478876
BC00372=478876
BC00373=478876
BC00374=478876
BC00375=478876
BC00376=478876
BC00377=478876
BC00378=478876
BC00379=478876
BC00380=478876
BC00381=478876
BC00382=478876
BC00383=478876
BC00384=480759
BC00385=480759
BC00386=560395
BC00387=606256
BC00388=606256
BC00389=606252
BC00390=606252
BC00391=606252
BC00392=606252
BC00393=654662
BC00394=654618
BC00395=654618
BC00396=654618
BC00397=654618
BC00398=654618
BC00399=654618
BC00400=654618
BC00401=654618
BC00402=654618
BC00403=654618
BC00404=686402
BC00405=686402
BC00406=686350
BC00407=686350
BC00408=686402
BC00409=652163
BC00410=658505
BC00411=725268
BC00412=747845
BC00413=747845
BC00414=747793
BC00415=747793
BC00416=747845
BC00417=778568
BC00418=778568
BC00419=778516
BC00420=778516
BC00421=758291
BC00422=652574
BC00423=652574
BC00424=774850
BC00425=784046
BC00426=784046
BC00427=784046
BC00428=784046
BC00429=784046
BC00430=784046
BC00431=784046
BC00432=784046
BC00433=784046
BC00434=784046
BC00435=784046
BC00436=821134
BC00437=821134
BC00438=821134
BC00439=821134
BC00440=821134
BC00441=821134
BC00442=821134
BC00443=821134
BC00444=821134
BC00445=821134
BC00446=728968
BC00447=735310
BC00448=802073
BC00449=802073
BC00450=802073
BC00451=802073
BC00452=802073
BC00453=802073
BC00454=817725
BC00455=657110
BC00456=380737
BC00457=417754
BC00458=467540
BC00459=497868
BC00460=497868
BC00461=535759
BC00462=535759
BC00463=535757
BC00464=535757
BC00465=535757
BC00466=535757
BC00467=535757
BC00468=485653
BC00469=485653
BC00470=485653
BC00471=485653
BC00472=485653
BC00473=485653
BC00474=485653
BC00475=485653
BC00476=485653
BC00477=485653
BC00478=485653
BC00479=485653
BC00480=485653
BC00481=485653
BC00482=601945
BC00483=615112
BC00484=615112
BC00485=615112
BC00486=615112
BC00487=615112
BC00488=615112
BC00489=615112
BC00490=615112
BC00491=615112
BC00492=615112
BC00493=615112
BC00494=615112
BC00495=615112
BC00496=615112
BC00497=615112
BC00498=615112
BC00499=615112
BC00500=658076
BC00501=658076
BC00502=658076
BC00503=658076
BC00504=658076
BC00505=659255
BC00506=747542
BC00507=715104
BC00508=719519
BC00509=719519
BC00510=719519
BC00511=719519
BC00512=719519
BC00513=757922
BC00514=750242
BC00515=750242
BC00516=750242
BC00517=714613
BC00518=655680
BC00519=655680
BC00520=765678
BC00521=799070
BC00522=799070
BC00523=799070
BC00524=799070
BC00525=799070
BC00526=799070
BC00527=799070
BC00528=799070
BC00529=799070
BC00530=799070
BC00531=799070
BC00532=799070
BC00533=799070
BC00534=799070
BC00535=799070
BC00536=799070
BC00537=845667
BC00538=845667
BC00539=845667
BC00540=845667
BC00541=845667
BC00542=736060
BC00543=824347
BC00544=791909
BC00545=791909
BC00546=791909
BC00547=791909
BC00548=791909
BC00549=791909
BC00550=757230
BC00551=501158
BC00552=467225
BC00553=513669
BC00554=494109
BC00555=467540
BC00556=467540
BC00557=478876
BC00558=478876
BC00559=478876
BC00560=478876
BC00561=478876
BC00562=478876
BC00563=478876
BC00564=478876
BC00565=478876
BC00566=478876
BC00567=478876
BC00568=478876
BC00569=479530
BC00570=502776
BC00571=571156
BC00572=606256
BC00573=606256
BC00574=606252
BC00575=606252
BC00576=606252
BC00577=654662
BC00578=654618
BC00579=654618
BC00580=654618
BC00581=654618
BC00582=654618
BC00583=654618
BC00584=654618
BC00585=654618
BC00586=686402
BC00587=686402
BC00588=686402
BC00589=686402
BC00590=643850
BC00591=700434
BC00592=737819
BC00593=747845
BC00594=747845
BC00595=747845
BC00596=747845
BC00597=773208
BC00598=778568
BC00599=778568
BC00600=751097
BC00601=652574
BC00602=654591
BC00603=763025
BC00604=784046
BC00605=784046
BC00606=784046
BC00607=784046
BC00608=784046
BC00609=784046
BC00610=784043
BC00611=784043
BC00612=784046
BC00613=821134
BC00614=821134
BC00615=821134
BC00616=821134
BC00617=821134
BC00618=821134
BC00619=821134
BC00620=821134
BC00621=720655
BC00622=777239
BC00623=814624
BC00624=820210
BC00625=810577
BC00626=810577
BC00627=810577
BC00628=810577
BC00629=823729
BC00630=823729
BC00631=813320
BC00632=702447
BC00633=426820
BC00634=509920
BC00635=467540
BC00636=467540
BC00637=467540
BC00638=521167
BC00639=520352
BC00640=535759
BC00641=535759
BC00642=535757
BC00643=535757
BC00644=535757
BC00645=535757
BC00646=485653
BC00647=485653
BC00648=485653
BC00649=485653
BC00650=485653
BC00651=485653
BC00652=485653
BC00653=485653
BC00654=485653
BC00655=485653
BC00656=485653
BC00657=600333
BC00658=615112
BC00659=615112
BC00660=615112
BC00661=615112
BC00662=615112
BC00663=615112
BC00664=615112
BC00665=615112
BC00666=615112
BC00667=615112
BC00668=615112
BC00669=615112
BC00670=615112
BC00671=615112
BC00672=658076
BC00673=658076
BC00674=658076
BC00675=658076
BC00676=645644
BC00677=726059
BC00678=715104
BC00679=719519
BC00680=719519
BC00681=719519
BC00682=719519
BC00683=750242
BC00684=750242
BC00685=750242
BC00686=722045
BC00687=655680
BC00688=656245
BC00689=762546
BC00690=762546
BC00691=799070
BC00692=799070
BC00693=799070
BC00694=799070
BC00695=799070
BC00696=799070
BC00697=799070
BC00698=799070
BC00699=799070
BC00700=799070
BC00701=799070
BC00702=799070
BC00703=799070
BC00704=845667
BC00705=845667
BC00706=845667
BC00707=845667
BC00708=722449
BC00709=802864
BC00710=791909
BC00711=791909
BC00712=807068
BC00713=807068
BC00714=807068
BC00715=807068
BC00716=807068
BC00717=807068
BC00718=807068
BC00719=799597
BC00720=784137
BC00721=739235
BC00722=639407
///POSTYPE BASE
///RECTAN
///RCONF 0,0,0,0,0,0,0,0,0,0,0,0,0,0,0,0,0,0,0,0,0,0,0,0
P00006=-2.449,0.031,8.825,0.0000,0.0000,0.0000
P00056=0.000,0.000,5.000,0.0000,0.0000,0.0000
P00301=0.005,-4.708,-4.628,0.0000,0.0000,0.0000
P00302=0.052,-2.937,-4.426,0.0000,0.0000,0.0000
P00303=-0.004,-1.437,-4.584,0.0000,0.0000,0.0000
P00304=0.028,-1.666,-4.234,0.0000,0.0000,0.0000
P00305=-0.003,-1.920,-3.501,0.0000,0.0000,0.0000
P00306=0.015,-2.252,-3.054,0.0000,0.0000,0.0000
P00307=0.019,-2.151,-5.077,0.0000,0.0000,0.0000
P00308=-0.003,-2.092,-4.888,0.0000,0.0000,0.0000
P00309=-0.040,-2.205,-4.992,0.0000,0.0000,0.0000
P00310=-0.006,-2.490,-5.925,0.0000,0.0000,0.0000
P00311=-0.007,-2.079,-5.307,0.0000,0.0000,0.0000
P00312=-0.032,2.202,-7.632,0.0000,0.0000,0.0000
P00351=13.563,-0.027,-0.653,0.0000,0.0000,0.0000
P00352=13.252,-0.027,-0.827,0.0000,0.0000,0.0000
P00353=10.971,-0.082,0.776,0.0000,0.0000,0.0000
P00354=-0.024,2.508,-1.824,0.0000,0.0000,0.0000
P00355=-0.001,2.528,-1.131,0.0000,0.0000,0.0000
P00356=-0.034,2.921,-0.262,0.0000,0.0000,0.0000
P00357=0.003,3.386,-0.091,0.0000,0.0000,0.0000
P00358=0.014,3.037,-0.020,0.0000,0.0000,0.0000
P00359=-0.005,2.731,0.912,0.0000,0.0000,0.0000
P00360=-0.011,3.412,0.438,0.0000,0.0000,0.0000
P00361=0.018,3.050,1.253,0.0000,0.0000,0.0000
P00362=0.014,2.784,0.148,0.0000,0.0000,0.0000
//INST
///DATE 2025/04/10 12:04
///ATTR SC,RW
///GROUP1 RB1,BS1
NOP
CALL JOB:MOVE_INTO_TUNNEL
MOVJ C00000 BC00000 VJ=10.00
MOVJ C00001 BC00001 VJ=10.00
MOVJ C00002 BC00002 VJ=10.00
MOVJ C00003 BC00003 VJ=10.00
MOVJ C00004 BC00004 VJ=10.00
'------------------------
'W29.2
'------------------------
MOVL C00005 BC00005 V=500.0
'------------------------
'W63.5
'------------------------
SFTOF
MOVL C00006 BC00006 V=166.7 PL=0
REFP 3 C00007 BC00007
CALL JOB:SEARCH-R1
IMOV P0056 V=50.0 PL=0
SET P0301 P0006
SFTON P0301
REFP 3 C00008 BC00008
CALL JOB:SEARCH-R1
SET P0301 P0006
SFTON P0301
MOVL C00009 BC00009 V=166.7 PL=0
SFTOF
MOVL C00010 BC00010 V=500.0
MOVL C00011 BC00011 V=166.7 PL=0
REFP 3 C00012 BC00012
CALL JOB:SEARCH-R1
IMOV P0056 V=50.0 PL=0
SET P0302 P0006
SFTON P0302
REFP 3 C00013 BC00013
CALL JOB:SEARCH-R1
SET P0302 P0006
SFTON P0302
MOVL C00014 BC00014 V=166.7 PL=0
SFTOF
MOVL C00015 BC00015 V=500.0
MOVL C00016 BC00016 V=166.7 PL=0
REFP 3 C00017 BC00017
CALL JOB:SEARCH-R1
IMOV P0056 V=50.0 PL=0
SET P0303 P0006
SFTON P0303
REFP 3 C00018 BC00018
CALL JOB:SEARCH-R1
SET P0303 P0006
SFTON P0303
SFTOF
MOVL C00019 BC00019 V=166.7 PL=0
MOVL C00020 BC00020 V=500.0
MOVJ C00021 BC00021 VJ=30.00
MOVJ C00022 BC00022 VJ=30.00
MOVJ C00023 BC00023 VJ=30.00
MOVL C00024 BC00024 V=500.0
'------------------------
'W29.14
'------------------------
MOVL C00025 BC00025 V=166.7 PL=0
REFP 3 C00026 BC00026
CALL JOB:SEARCH-R1
IMOV P0056 V=23.0 PL=0
SET P0304 P0006
SFTON P0304
REFP 3 C00027 BC00027
CALL JOB:SEARCH-R1
SET P0304 P0006
SFTON P0304
MOVL C00028 BC00028 V=66.7 PL=0
SFTOF
'PRZEJAZD
MOVL C00029 BC00029 V=500.0
MOVL C00030 BC00030 V=500.0
'------------------------
'W63.17
'------------------------
MOVL C00031 BC00031 V=166.7 PL=0
REFP 3 C00032 BC00032
CALL JOB:SEARCH-R1
IMOV P0056 V=23.0 PL=0
SET P0305 P0006
SFTON P0305
REFP 3 C00033 BC00033
CALL JOB:SEARCH-R1
SET P0305 P0006
SFTON P0305
MOVL C00034 BC00034 V=166.7 PL=0
SFTOF
MOVL C00035 BC00035 V=500.0
MOVL C00036 BC00036 V=166.7
REFP 3 C00037 BC00037
CALL JOB:SEARCH-R1
IMOV P0056 V=23.0 PL=0
SET P0306 P0006
SFTON P0306
REFP 3 C00038 BC00038
CALL JOB:SEARCH-R1
SET P0306 P0006
SFTON P0306
MOVL C00039 BC00039 V=166.7 PL=0
'PRZEJAZD
MOVL C00040 BC00040 V=500.0
MOVL C00041 BC00041 V=166.7
REFP 3 C00042 BC00042
CALL JOB:SEARCH-R1
IMOV P0056 V=23.0 PL=0
SET P0307 P0006
SFTON P0307
REFP 3 C00043 BC00043
CALL JOB:SEARCH-R1
SET P0307 P0006
SFTON P0307
MOVL C00044 BC00044 V=166.7 PL=0
SFTOF
MOVL C00045 BC00045 V=500.0
MOVL C00046 BC00046 V=500.0
MOVL C00047 BC00047 V=333.3
MOVL C00048 BC00048 V=500.0
MOVL C00049 BC00049 V=166.7
REFP 3 C00050 BC00050
CALL JOB:SEARCH-R1
IMOV P0056 V=23.0 PL=0
SET P0308 P0006
SFTON P0308
REFP 3 C00051 BC00051
CALL JOB:SEARCH-R1
SET P0308 P0006
SFTON P0308
MOVL C00052 BC00052 V=166.7 PL=0
SFTOF
MOVL C00053 BC00053 V=500.0
MOVL C00054 BC00054 V=166.7
REFP 3 C00055 BC00055
CALL JOB:SEARCH-R1
IMOV P0056 V=23.0 PL=0
SET P0309 P0006
SFTON P0309
REFP 3 C00056 BC00056
CALL JOB:SEARCH-R1
SET P0309 P0006
SFTON P0309
MOVL C00057 BC00057 V=500.0 PL=0
SFTOF
COMM PAUSE
COMM MOVJ C00058 BC00058 VJ=20.00
COMM MOVJ C00059 BC00059 VJ=20.00
COMM MOVJ C00060 BC00060 VJ=30.00
COMM MOVJ C00061 BC00061 VJ=30.00
COMM MOVJ C00062 BC00062 VJ=30.00
COMM MOVL C00063 BC00063 V=500.0
COMM '------------------------
COMM 'W63.20
COMM '------------------------
COMM MOVL C00064 BC00064 V=166.7 PL=0
COMM REFP 3 C00065 BC00065
COMM CALL JOB:SEARCH-R1
COMM IMOV P0056 V=23.0 PL=0
COMM SET P0308 P0006
COMM SFTON P0308
COMM REFP 3 C00066 BC00066
COMM CALL JOB:SEARCH-R1
COMM SET P0308 P0006
COMM SFTON P0308
COMM MOVL C00067 BC00067 V=166.7 PL=0
COMM SFTOF
COMM PAUSE
COMM 'PRZEJAZD
COMM MOVL C00068 BC00068 V=500.0
COMM '------------------------
COMM 'W63.23
COMM '------------------------
COMM MOVL C00069 BC00069 V=166.7 PL=0
COMM REFP 3 C00070 BC00070
COMM CALL JOB:SEARCH-R1
COMM IMOV P0056 V=23.0 PL=0
COMM SET P0309 P0006
COMM SFTON P0309
COMM REFP 3 C00071 BC00071
COMM CALL JOB:SEARCH-R1
COMM SET P0309 P0006
COMM SFTON P0309
COMM MOVL C00072 BC00072 V=250.0 PL=0
COMM SFTOF
COMM MOVL C00073 BC00073 V=500.0
COMM MOVL C00074 BC00074 V=166.7 PL=0
COMM REFP 3 C00075 BC00075
COMM CALL JOB:SEARCH-R1
COMM IMOV P0056 V=23.0 PL=0
COMM SET P0310 P0006
COMM SFTON P0310
COMM REFP 3 C00076 BC00076
COMM CALL JOB:SEARCH-R1
COMM SET P0310 P0006
COMM SFTON P0310
COMM MOVL C00077 BC00077 V=250.0 PL=0
COMM SFTOF
COMM MOVL C00078 BC00078 V=500.0
COMM MOVL C00079 BC00079 V=166.7 PL=0
COMM REFP 3 C00080 BC00080
COMM CALL JOB:SEARCH-R1
COMM IMOV P0056 V=23.0 PL=0
COMM SET P0311 P0006
COMM SFTON P0311
COMM REFP 3 C00081 BC00081
COMM CALL JOB:SEARCH-R1
COMM SET P0311 P0006
COMM SFTON P0311
COMM MOVL C00082 BC00082 V=250.0 PL=0
COMM SFTOF
MOVL C00083 BC00083 V=500.0
MOVL C00084 BC00084 V=500.0
MOVL C00085 BC00085 V=333.3
'------------------------
'W29.29
'------------------------
MOVL C00086 BC00086 V=166.7 PL=0
REFP 3 C00087 BC00087
CALL JOB:SEARCH-R1
IMOV P0056 V=23.0 PL=0
SET P0312 P0006
SFTON P0312
REFP 3 C00088 BC00088
CALL JOB:SEARCH-R1
SET P0312 P0006
SFTON P0312
MOVL C00089 BC00089 V=250.0 PL=0
SFTOF
'PRZEJAZD
MOVL C00090 BC00090 V=333.3
'PRZEJAZD
MOVJ C00091 BC00091 VJ=30.00
MOVJ C00092 BC00092 VJ=20.00
MOVJ C00093 BC00093 VJ=50.00
MOVJ C00094 BC00094 VJ=20.00
MOVJ C00095 BC00095 VJ=10.00
MOVJ C00096 BC00096 VJ=20.00
MOVJ C00097 BC00097 VJ=20.00
'------------------------
'W28.2
'------------------------
MOVJ C00098 BC00098 VJ=10.00
MOVJ C00099 BC00099 VJ=10.00
MOVL C00100 BC00100 V=500.0
MOVL C00101 BC00101 V=500.0
'------------------------
'W62.5
'------------------------
MOVL C00102 BC00102 V=166.7 PL=0
REFP 3 C00103 BC00103
CALL JOB:SEARCH-R1
IMOV P0056 V=23.0 PL=0
SET P0351 P0006
SFTON P0351
REFP 3 C00104 BC00104
CALL JOB:SEARCH-R1
SET P0351 P0006
SFTON P0351
MOVL C00105 BC00105 V=250.0 PL=0
SFTOF
'PRZEJAZD
MOVL C00106 BC00106 V=500.0
MOVL C00107 BC00107 V=500.0
MOVL C00108 BC00108 V=500.0
MOVL C00109 BC00109 V=166.7 PL=0
REFP 3 C00110 BC00110
CALL JOB:SEARCH-R1
IMOV P0056 V=23.0 PL=0
SET P0352 P0006
SFTON P0352
REFP 3 C00111 BC00111
CALL JOB:SEARCH-R1
SET P0352 P0006
SFTON P0352
MOVL C00112 BC00112 V=250.0 PL=0
SFTOF
MOVL C00113 BC00113 V=500.0
'------------------------
'W29.8
'------------------------
MOVL C00114 BC00114 V=166.7 PL=0
REFP 3 C00115 BC00115
CALL JOB:SEARCH-R1
IMOV P0056 V=23.0 PL=0
SET P0353 P0006
SFTON P0353
REFP 3 C00116 BC00116
CALL JOB:SEARCH-R1
SET P0353 P0006
SFTON P0353
MOVL C00117 BC00117 V=250.0 PL=0
SFTOF
MOVL C00118 BC00118 V=500.0
'PRZEJAZD
MOVL C00119 BC00119 V=500.0
MOVJ C00120 BC00120 VJ=20.00
MOVL C00121 BC00121 V=500.0
MOVL C00122 BC00122 V=500.0
MOVL C00123 BC00123 V=500.0
'------------------------
'W29.11
'------------------------
MOVL C00124 BC00124 V=166.7 PL=0
REFP 3 C00125 BC00125
CALL JOB:SEARCH-R1
IMOV P0056 V=23.0 PL=0
SET P0354 P0006
SFTON P0354
REFP 3 C00126 BC00126
CALL JOB:SEARCH-R1
SET P0354 P0006
SFTON P0354
MOVL C00127 BC00127 V=250.0 PL=0
SFTOF
'PRZEJAZD
MOVL C00128 BC00128 V=500.0
'------------------------
'W29.14
'------------------------
MOVL C00129 BC00129 V=166.7 PL=0
REFP 3 C00130 BC00130
CALL JOB:SEARCH-R1
IMOV P0056 V=23.0 PL=0
SET P0355 P0006
SFTON P0355
REFP 3 C00131 BC00131
CALL JOB:SEARCH-R1
SET P0355 P0006
SFTON P0355
MOVL C00132 BC00132 V=250.0 PL=0
SFTOF
'PRZEJAZD
MOVL C00133 BC00133 V=500.0
'------------------------
'W63.17
'------------------------
MOVL C00134 BC00134 V=166.7 PL=0
REFP 3 C00135 BC00135
CALL JOB:SEARCH-R1
IMOV P0056 V=23.0 PL=0
SET P0356 P0006
SFTON P0356
REFP 3 C00136 BC00136
CALL JOB:SEARCH-R1
SET P0356 P0006
SFTON P0356
MOVL C00137 BC00137 V=250.0 PL=0
SFTOF
MOVL C00138 BC00138 V=500.0
MOVL C00139 BC00139 V=166.7 PL=0
REFP 3 C00140 BC00140
CALL JOB:SEARCH-R1
IMOV P0056 V=23.0 PL=0
SET P0357 P0006
SFTON P0357
REFP 3 C00141 BC00141
CALL JOB:SEARCH-R1
SET P0357 P0006
SFTON P0357
MOVL C00142 BC00142 V=250.0 PL=0
SFTOF
MOVL C00143 BC00143 V=500.0
MOVJ C00144 BC00144 VJ=10.00
MOVL C00145 BC00145 V=416.7
MOVL C00146 BC00146 V=500.0
MOVL C00147 BC00147 V=166.7 PL=0
REFP 3 C00148 BC00148
CALL JOB:SEARCH-R1
IMOV P0056 V=23.0 PL=0
SET P0358 P0006
SFTON P0358
REFP 3 C00149 BC00149
CALL JOB:SEARCH-R1
SET P0358 P0006
SFTON P0358
MOVL C00150 BC00150 V=250.0 PL=0
SFTOF
MOVL C00151 BC00151 V=500.0
MOVL C00152 BC00152 V=166.7 PL=0
REFP 3 C00153 BC00153
CALL JOB:SEARCH-R1
IMOV P0056 V=23.0 PL=0
SET P0359 P0006
SFTON P0359
REFP 3 C00154 BC00154
CALL JOB:SEARCH-R1
SET P0359 P0006
SFTON P0359
MOVL C00155 BC00155 V=250.0 PL=0
SFTOF
COMM 'PRZEJAZD
COMM MOVL C00156 BC00156 V=500.0
COMM MOVJ C00157 BC00157 VJ=30.00
COMM MOVJ C00158 BC00158 VJ=30.00
COMM MOVJ C00159 BC00159 VJ=30.00
COMM MOVL C00160 BC00160 V=500.0
COMM MOVL C00161 BC00161 V=500.0
COMM '------------------------
COMM 'W62.20
COMM '------------------------
COMM MOVL C00162 BC00162 V=166.7 PL=0
COMM REFP 3 C00163 BC00163
COMM CALL JOB:SEARCH-R1
COMM IMOV P0056 V=23.0 PL=0
COMM SET P0358 P0006
COMM SFTON P0358
COMM REFP 3 C00164 BC00164
COMM CALL JOB:SEARCH-R1
COMM SET P0358 P0006
COMM SFTON P0358
COMM MOVL C00165 BC00165 V=250.0 PL=0
COMM SFTOF
COMM 'PRZEJAZD
COMM MOVL C00166 BC00166 V=500.0
COMM '------------------------
COMM 'W63.23
COMM '------------------------
COMM MOVL C00167 BC00167 V=166.7 PL=0
COMM REFP 3 C00168 BC00168
COMM CALL JOB:SEARCH-R1
COMM IMOV P0056 V=23.0 PL=0
COMM SET P0359 P0006
COMM SFTON P0359
COMM REFP 3 C00169 BC00169
COMM CALL JOB:SEARCH-R1
COMM SET P0359 P0006
COMM SFTON P0359
COMM MOVL C00170 BC00170 V=250.0 PL=0
COMM MOVL C00171 BC00171 V=500.0
COMM '------------------------
COMM 'W29.29
COMM '------------------------
COMM MOVL C00172 BC00172 V=166.7 PL=0
COMM REFP 3 C00173 BC00173
COMM CALL JOB:SEARCH-R1
COMM IMOV P0056 V=23.0 PL=0
COMM SET P0360 P0006
COMM SFTON P0360
COMM REFP 3 C00174 BC00174
COMM CALL JOB:SEARCH-R1
COMM SET P0360 P0006
COMM SFTON P0360
COMM MOVL C00175 BC00175 V=250.0 PL=0
COMM SFTOF
COMM 'PRZEJAZD
COMM MOVL C00176 BC00176 V=500.0
COMM MOVL C00177 BC00177 V=166.7 PL=0
COMM REFP 3 C00178 BC00178
COMM CALL JOB:SEARCH-R1
COMM IMOV P0056 V=23.0 PL=0
COMM SET P0361 P0006
COMM SFTON P0361
COMM REFP 3 C00179 BC00179
COMM CALL JOB:SEARCH-R1
COMM SET P0361 P0006
COMM SFTON P0361
COMM MOVL C00180 BC00180 V=250.0 PL=0
COMM SFTOF
COMM '------------------------
COMM 'W29.32
COMM '------------------------
COMM 'PRZEJAZD
MOVL C00181 BC00181 V=500.0
MOVJ C00182 BC00182 VJ=10.00
MOVL C00183 BC00183 V=416.7
MOVL C00184 BC00184 V=166.7 PL=0
REFP 3 C00185 BC00185
CALL JOB:SEARCH-R1
IMOV P0056 V=23.0 PL=0
SET P0362 P0006
SFTON P0362
REFP 3 C00186 BC00186
CALL JOB:SEARCH-R1
SET P0362 P0006
SFTON P0362
MOVL C00187 BC00187 V=250.0 PL=0
SFTOF
MOVJ C00188 BC00188 VJ=20.00
MOVJ C00189 BC00189 VJ=30.00
MOVJ C00190 BC00190 VJ=30.00
'KONIEC SEARCH WEW STRONA
MOVJ C00191 BC00191 VJ=30.00
MOVJ C00192 BC00192 VJ=20.00
MOVJ C00193 BC00193 VJ=10.00
MOVJ C00194 BC00194 VJ=20.00
MOVJ C00195 BC00195 VJ=20.00
'------------------------
'W29.2
'------------------------
MOVL C00196 BC00196 V=500.0
'------------------------
'W63.5
MACRO1 MJ#(0) ARGF9
'------------------------
SFTOF
SFTON P0301
MOVL C00197 BC00197 V=166.7 PL=0
ARCON
MOVL C00198 BC00198 V=10.0
ARCOF
SFTOF
MOVL C00199 BC00199 V=500.0
SFTON P0302
MOVL C00200 BC00200 V=166.7 PL=0
ARCON
MOVL C00201 BC00201 V=10.0
ARCOF
MOVL C00202 BC00202 V=166.7 PL=0
SFTOF
MOVL C00203 BC00203 V=500.0
SFTON P0303
MOVL C00204 BC00204 V=166.7 PL=0
ARCON
MOVL C00205 BC00205 V=10.0
ARCOF
SFTOF
MOVL C00206 BC00206 V=166.7 PL=0
MOVL C00207 BC00207 V=500.0
MOVJ C00208 BC00208 VJ=30.00
MOVJ C00209 BC00209 VJ=30.00
MOVJ C00210 BC00210 VJ=30.00
MOVL C00211 BC00211 V=500.0
'------------------------
'W29.14
'------------------------
SFTON P0304
MOVL C00212 BC00212 V=166.7 PL=0
ARCON
MOVL C00213 BC00213 V=10.0
ARCOF
MOVL C00214 BC00214 V=166.7 PL=0
SFTOF
'PRZEJAZD
MOVL C00215 BC00215 V=500.0
MOVL C00216 BC00216 V=500.0
'------------------------
'W63.17
'------------------------
SFTON P0305
MOVL C00217 BC00217 V=166.7 PL=0
ARCON
MOVL C00218 BC00218 V=10.0
ARCOF
MOVL C00219 BC00219 V=166.7 PL=0
SFTOF
MOVL C00220 BC00220 V=500.0
SFTON P0306
MOVL C00221 BC00221 V=166.7
ARCON
MOVL C00222 BC00222 V=10.0
ARCOF
MOVL C00223 BC00223 V=166.7 PL=0
SFTOF
'PRZEJAZD
MOVL C00224 BC00224 V=500.0
SFTON P0307
MOVL C00225 BC00225 V=166.7
ARCON
MOVL C00226 BC00226 V=10.0
ARCOF
MOVL C00227 BC00227 V=166.7 PL=0
SFTOF
MOVL C00228 BC00228 V=500.0
MOVL C00229 BC00229 V=500.0
MOVL C00230 BC00230 V=333.3
MOVL C00231 BC00231 V=250.0
MOVL C00232 BC00232 V=500.0
SFTON P0308
MOVL C00233 BC00233 V=166.7
ARCON
MOVL C00234 BC00234 V=10.0
ARCOF
MOVL C00235 BC00235 V=166.7 PL=0
SFTOF
MOVL C00236 BC00236 V=500.0
SFTON P0309
MOVL C00237 BC00237 V=166.7
ARCON
MOVL C00238 BC00238 V=10.0
ARCOF
MOVL C00239 BC00239 V=500.0 PL=0
SFTOF
COMM PAUSE
COMM MOVJ C00240 BC00240 VJ=20.00
COMM MOVJ C00241 BC00241 VJ=20.00
COMM MOVJ C00242 BC00242 VJ=30.00
COMM MOVJ C00243 BC00243 VJ=30.00
COMM MOVJ C00244 BC00244 VJ=30.00
COMM MOVL C00245 BC00245 V=500.0
COMM '------------------------
COMM 'W63.20
COMM '------------------------
COMM SFTON P0308
COMM MOVL C00246 BC00246 V=166.7 PL=0
COMM ARCON
COMM MOVL C00247 BC00247 V=10.0
COMM ARCOF
COMM MOVL C00248 BC00248 V=166.7 PL=0
COMM SFTOF
COMM 'PRZEJAZD
COMM MOVL C00249 BC00249 V=500.0
COMM '------------------------
COMM 'W63.23
COMM '------------------------
COMM SFTON P0309
COMM MOVL C00250 BC00250 V=166.7 PL=0
COMM ARCON
COMM MOVL C00251 BC00251 V=10.0
COMM ARCOF
COMM MOVL C00252 BC00252 V=250.0 PL=0
COMM SFTOF
COMM MOVL C00253 BC00253 V=500.0
COMM SFTON P0310
COMM MOVL C00254 BC00254 V=166.7 PL=0
COMM ARCON
COMM MOVL C00255 BC00255 V=10.0
COMM ARCOF
COMM MOVL C00256 BC00256 V=250.0 PL=0
COMM SFTOF
COMM MOVL C00257 BC00257 V=500.0
COMM SFTON P0311
COMM MOVL C00258 BC00258 V=166.7 PL=0
COMM ARCON
COMM MOVL C00259 BC00259 V=10.0
COMM ARCOF
COMM MOVL C00260 BC00260 V=250.0 PL=0
SFTOF
MOVL C00261 BC00261 V=500.0
MOVL C00262 BC00262 V=500.0
MOVL C00263 BC00263 V=333.3
MOVL C00264 BC00264 V=250.0
'------------------------
'W29.29
'------------------------
SFTON P0312
COMM MOVL C00265 BC00265 V=166.7 PL=0
COMM ARCON
COMM MOVL C00266 BC00266 V=9.2
COMM ARCOF
MOVL C00267 BC00267 V=250.0 PL=0
MOVL C00268 BC00268 V=333.3 PL=0
ARCON
MOVL C00269 BC00269 V=9.2
ARCOF
SFTOF
'PRZEJAZD
MOVL C00270 BC00270 V=333.3
MOVJ C00271 BC00271 VJ=30.00
MOVJ C00272 BC00272 VJ=20.00
MOVJ C00273 BC00273 VJ=50.00
MOVJ C00274 BC00274 VJ=20.00
MOVJ C00275 BC00275 VJ=10.00
MOVJ C00276 BC00276 VJ=20.00
MOVJ C00277 BC00277 VJ=20.00
'------------------------
'W28.2
'------------------------
MOVJ C00278 BC00278 VJ=10.00
MOVJ C00279 BC00279 VJ=10.00
MOVL C00280 BC00280 V=500.0
MOVL C00281 BC00281 V=500.0
'------------------------
'W62.5
'------------------------
SFTON P0351
MOVL C00282 BC00282 V=166.7 PL=0
ARCON
MOVL C00283 BC00283 V=10.0
ARCOF
MOVL C00284 BC00284 V=250.0 PL=0
SFTOF
'PRZEJAZD
MOVL C00285 BC00285 V=500.0
MOVL C00286 BC00286 V=500.0
MOVL C00287 BC00287 V=500.0
SFTON P0352
MOVL C00288 BC00288 V=166.7 PL=0
ARCON
MOVL C00289 BC00289 V=10.0
ARCOF
MOVL C00290 BC00290 V=250.0 PL=0
SFTOF
MOVL C00291 BC00291 V=500.0
'------------------------
'W29.8
'------------------------
SFTON P0353
MOVL C00292 BC00292 V=166.7 PL=0
ARCON
MOVL C00293 BC00293 V=10.0
ARCOF
MOVL C00294 BC00294 V=250.0 PL=0
SFTOF
MOVL C00295 BC00295 V=500.0
'PRZEJAZD
MOVL C00296 BC00296 V=500.0
MOVJ C00297 BC00297 VJ=20.00
MOVL C00298 BC00298 V=500.0
MOVL C00299 BC00299 V=500.0
MOVL C00300 BC00300 V=500.0
'------------------------
'W29.11
'------------------------
SFTON P0354
MOVL C00301 BC00301 V=166.7 PL=0
ARCON
MOVL C00302 BC00302 V=10.0
ARCOF
MOVL C00303 BC00303 V=250.0 PL=0
SFTOF
'PRZEJAZD
MOVL C00304 BC00304 V=500.0
'------------------------
'W29.14
'------------------------
SFTON P0355
MOVL C00305 BC00305 V=166.7 PL=0
ARCON
MOVL C00306 BC00306 V=10.0
ARCOF
MOVL C00307 BC00307 V=250.0 PL=0
SFTOF
'PRZEJAZD
MOVL C00308 BC00308 V=500.0
'------------------------
'W63.17
'------------------------
SFTON P0356
MOVL C00309 BC00309 V=166.7 PL=0
ARCON
MOVL C00310 BC00310 V=10.0
ARCOF
MOVL C00311 BC00311 V=250.0 PL=0
SFTOF
MOVL C00312 BC00312 V=500.0
SFTON P0357
MOVL C00313 BC00313 V=166.7 PL=0
ARCON
MOVL C00314 BC00314 V=10.0
ARCOF
MOVL C00315 BC00315 V=250.0 PL=0
SFTOF
MOVL C00316 BC00316 V=500.0
MOVJ C00317 BC00317 VJ=10.00
MOVL C00318 BC00318 V=416.7
MOVL C00319 BC00319 V=500.0
SFTON P0358
MOVL C00320 BC00320 V=166.7 PL=0
ARCON
MOVL C00321 BC00321 V=10.0
ARCOF
MOVL C00322 BC00322 V=250.0 PL=0
SFTOF
MOVL C00323 BC00323 V=500.0
SFTON P0359
MOVL C00324 BC00324 V=166.7 PL=0
ARCON
MOVL C00325 BC00325 V=10.0
ARCOF
MOVL C00326 BC00326 V=250.0 PL=0
SFTOF
COMM PAUSE
COMM 'PRZEJAZD
COMM MOVL C00327 BC00327 V=500.0
COMM MOVJ C00328 BC00328 VJ=30.00
COMM MOVJ C00329 BC00329 VJ=30.00
COMM MOVJ C00330 BC00330 VJ=30.00
COMM MOVL C00331 BC00331 V=500.0
COMM MOVL C00332 BC00332 V=500.0
COMM '------------------------
COMM 'W62.20
COMM '------------------------
COMM SFTON P0358
COMM MOVL C00333 BC00333 V=166.7 PL=0
COMM ARCON
COMM MOVL C00334 BC00334 V=10.0
COMM ARCOF
COMM MOVL C00335 BC00335 V=250.0 PL=0
COMM SFTOF
COMM 'PRZEJAZD
COMM MOVL C00336 BC00336 V=500.0
COMM '------------------------
COMM 'W63.23
COMM '------------------------
COMM SFTON P0359
COMM MOVL C00337 BC00337 V=166.7 PL=0
COMM ARCON
COMM MOVL C00338 BC00338 V=10.0
COMM ARCOF
COMM MOVL C00339 BC00339 V=250.0 PL=0
COMM MOVL C00340 BC00340 V=500.0
COMM '------------------------
COMM 'W29.29
COMM '------------------------
COMM SFTON P0360
COMM MOVL C00341 BC00341 V=166.7 PL=0
COMM ARCON
COMM MOVL C00342 BC00342 V=10.0
COMM ARCOF
COMM MOVL C00343 BC00343 V=250.0 PL=0
COMM SFTOF
COMM 'PRZEJAZD
COMM MOVL C00344 BC00344 V=500.0
COMM SFTON P0361
COMM MOVL C00345 BC00345 V=166.7 PL=0
COMM ARCON
COMM MOVL C00346 BC00346 V=10.0
COMM ARCOF
COMM MOVL C00347 BC00347 V=250.0 PL=0
SFTOF
'------------------------
'W29.32
'------------------------
'PRZEJAZD
MOVL C00348 BC00348 V=500.0
MOVJ C00349 BC00349 VJ=10.00
MOVL C00350 BC00350 V=416.7
SFTON P0362
COMM MOVL C00351 BC00351 V=166.7 PL=0
COMM ARCON
COMM MOVL C00352 BC00352 V=9.2
COMM ARCOF
COMM MOVL C00353 BC00353 V=250.0 PL=0
COMM MOVL C00354 BC00354 V=250.0
MOVL C00355 BC00355 V=166.7
ARCON
MOVL C00356 BC00356 V=9.2
ARCOF
SFTOF
MOVL C00357 BC00357 V=166.7
MOVJ C00358 BC00358 VJ=20.00
MOVJ C00359 BC00359 VJ=30.00
MOVJ C00360 BC00360 VJ=30.00
CALL JOB:MOVE_OUT_OF_TUNNEL
CALL JOB:CLEAN-R1
CALL JOB:MOVE_INTO_TUNNEL
'KONIEC SPAWANIA WEW STRONA
MOVJ C00361 BC00361 VJ=10.00
MOVJ C00362 BC00362 VJ=10.00
MOVJ C00363 BC00363 VJ=10.00
MOVJ C00364 BC00364 VJ=20.00
MOVJ C00365 BC00365 VJ=20.00
MOVJ C00366 BC00366 VJ=10.00
MOVJ C00367 BC00367 VJ=10.00
'------------------------
'W29.2
'------------------------
MOVL C00368 BC00368 V=500.0
'------------------------
'W63.5
'------------------------
SFTOF
MOVL C00369 BC00369 V=166.7 PL=0
REFP 3 C00370 BC00370
CALL JOB:SEARCH-R1
IMOV P0056 V=50.0 PL=0
SET P0301 P0006
SFTON P0301
REFP 3 C00371 BC00371
CALL JOB:SEARCH-R1
SET P0301 P0006
SFTON P0301
MOVL C00372 BC00372 V=166.7 PL=0
SFTOF
MOVL C00373 BC00373 V=500.0
MOVL C00374 BC00374 V=166.7 PL=0
REFP 3 C00375 BC00375
CALL JOB:SEARCH-R1
IMOV P0056 V=50.0 PL=0
SET P0302 P0006
SFTON P0302
REFP 3 C00376 BC00376
CALL JOB:SEARCH-R1
SET P0302 P0006
SFTON P0302
MOVL C00377 BC00377 V=166.7 PL=0
SFTOF
MOVL C00378 BC00378 V=500.0
MOVL C00379 BC00379 V=166.7 PL=0
REFP 3 C00380 BC00380
CALL JOB:SEARCH-R1
IMOV P0056 V=50.0 PL=0
SET P0303 P0006
SFTON P0303
REFP 3 C00381 BC00381
CALL JOB:SEARCH-R1
SET P0303 P0006
SFTON P0303
SFTOF
MOVL C00382 BC00382 V=166.7 PL=0
MOVL C00383 BC00383 V=500.0
MOVJ C00384 BC00384 VJ=30.00
MOVJ C00385 BC00385 VJ=30.00
MOVJ C00386 BC00386 VJ=20.00
MOVJ C00387 BC00387 VJ=30.00
MOVL C00388 BC00388 V=500.0
'------------------------
'W29.14
'------------------------
MOVL C00389 BC00389 V=166.7 PL=0
REFP 3 C00390 BC00390
CALL JOB:SEARCH-R1
IMOV P0056 V=23.0 PL=0
SET P0304 P0006
SFTON P0304
REFP 3 C00391 BC00391
CALL JOB:SEARCH-R1
SET P0304 P0006
SFTON P0304
MOVL C00392 BC00392 V=66.7 PL=0
SFTOF
'PRZEJAZD
MOVL C00393 BC00393 V=500.0
MOVL C00394 BC00394 V=500.0
'------------------------
'W63.17
'------------------------
MOVL C00395 BC00395 V=166.7 PL=0
REFP 3 C00396 BC00396
CALL JOB:SEARCH-R1
IMOV P0056 V=23.0 PL=0
SET P0305 P0006
SFTON P0305
REFP 3 C00397 BC00397
CALL JOB:SEARCH-R1
SET P0305 P0006
SFTON P0305
MOVL C00398 BC00398 V=166.7 PL=0
SFTOF
MOVL C00399 BC00399 V=500.0
MOVL C00400 BC00400 V=166.7
REFP 3 C00401 BC00401
CALL JOB:SEARCH-R1
IMOV P0056 V=23.0 PL=0
SET P0306 P0006
SFTON P0306
REFP 3 C00402 BC00402
CALL JOB:SEARCH-R1
SET P0306 P0006
SFTON P0306
MOVL C00403 BC00403 V=166.7 PL=0
'PRZEJAZD
MOVL C00404 BC00404 V=500.0
MOVL C00405 BC00405 V=166.7
REFP 3 C00406 BC00406
CALL JOB:SEARCH-R1
IMOV P0056 V=23.0 PL=0
SET P0307 P0006
SFTON P0307
REFP 3 C00407 BC00407
CALL JOB:SEARCH-R1
SET P0307 P0006
SFTON P0307
MOVL C00408 BC00408 V=166.7 PL=0
SFTOF
MOVL C00409 BC00409 V=500.0
MOVL C00410 BC00410 V=500.0
MOVL C00411 BC00411 V=333.3
MOVL C00412 BC00412 V=500.0
MOVL C00413 BC00413 V=166.7
REFP 3 C00414 BC00414
CALL JOB:SEARCH-R1
IMOV P0056 V=23.0 PL=0
SET P0308 P0006
SFTON P0308
REFP 3 C00415 BC00415
CALL JOB:SEARCH-R1
SET P0308 P0006
SFTON P0308
MOVL C00416 BC00416 V=166.7 PL=0
SFTOF
MOVL C00417 BC00417 V=500.0
MOVL C00418 BC00418 V=166.7
REFP 3 C00419 BC00419
CALL JOB:SEARCH-R1
IMOV P0056 V=23.0 PL=0
SET P0309 P0006
SFTON P0309
REFP 3 C00420 BC00420
CALL JOB:SEARCH-R1
SET P0309 P0006
SFTON P0309
MOVL C00421 BC00421 V=166.7 PL=0
SFTOF
COMM PAUSE
COMM MOVJ C00422 BC00422 VJ=20.00
COMM MOVJ C00423 BC00423 VJ=20.00
COMM MOVJ C00424 BC00424 VJ=30.00
COMM MOVJ C00425 BC00425 VJ=30.00
COMM MOVL C00426 BC00426 V=500.0
COMM '------------------------
COMM 'W63.20
COMM '------------------------
COMM MOVL C00427 BC00427 V=166.7 PL=0
COMM REFP 3 C00428 BC00428
COMM CALL JOB:SEARCH-R1
COMM IMOV P0056 V=23.0 PL=0
COMM SET P0308 P0006
COMM SFTON P0308
COMM REFP 3 C00429 BC00429
COMM CALL JOB:SEARCH-R1
COMM SET P0308 P0006
COMM SFTON P0308
COMM MOVL C00430 BC00430 V=166.7 PL=0
COMM SFTOF
COMM 'PRZEJAZD
COMM MOVL C00431 BC00431 V=500.0
COMM '------------------------
COMM 'W63.23
COMM '------------------------
COMM MOVL C00432 BC00432 V=166.7 PL=0
COMM REFP 3 C00433 BC00433
COMM CALL JOB:SEARCH-R1
COMM IMOV P0056 V=23.0 PL=0
COMM SET P0309 P0006
COMM SFTON P0309
COMM REFP 3 C00434 BC00434
COMM CALL JOB:SEARCH-R1
COMM SET P0309 P0006
COMM SFTON P0309
COMM MOVL C00435 BC00435 V=250.0 PL=0
COMM SFTOF
COMM MOVL C00436 BC00436 V=500.0
COMM MOVL C00437 BC00437 V=166.7 PL=0
COMM REFP 3 C00438 BC00438
COMM CALL JOB:SEARCH-R1
COMM IMOV P0056 V=23.0 PL=0
COMM SET P0310 P0006
COMM SFTON P0310
COMM REFP 3 C00439 BC00439
COMM CALL JOB:SEARCH-R1
COMM SET P0310 P0006
COMM SFTON P0310
COMM MOVL C00440 BC00440 V=250.0 PL=0
COMM SFTOF
COMM MOVL C00441 BC00441 V=500.0
COMM MOVL C00442 BC00442 V=166.7 PL=0
COMM REFP 3 C00443 BC00443
COMM CALL JOB:SEARCH-R1
COMM IMOV P0056 V=23.0 PL=0
COMM SET P0311 P0006
COMM SFTON P0311
COMM REFP 3 C00444 BC00444
COMM CALL JOB:SEARCH-R1
COMM SET P0311 P0006
COMM SFTON P0311
COMM MOVL C00445 BC00445 V=250.0 PL=0
SFTOF
MOVL C00446 BC00446 V=500.0
MOVL C00447 BC00447 V=500.0
MOVL C00448 BC00448 V=333.3
'------------------------
'W29.29
'------------------------
MOVL C00449 BC00449 V=250.0
MOVL C00450 BC00450 V=166.7 PL=0
REFP 3 C00451 BC00451
CALL JOB:SEARCH-R1
IMOV P0056 V=23.0 PL=0
SET P0312 P0006
SFTON P0312
REFP 3 C00452 BC00452
CALL JOB:SEARCH-R1
SET P0312 P0006
SFTON P0312
MOVL C00453 BC00453 V=250.0 PL=0
SFTOF
'PRZEJAZD
MOVL C00454 BC00454 V=333.3
'PRZEJAZD
MOVJ C00455 BC00455 VJ=20.00
MOVJ C00456 BC00456 VJ=50.00
MOVJ C00457 BC00457 VJ=20.00
MOVJ C00458 BC00458 VJ=10.00
'------------------------
'W28.2
'------------------------
MOVJ C00459 BC00459 VJ=10.00
MOVJ C00460 BC00460 VJ=10.00
MOVL C00461 BC00461 V=500.0
MOVL C00462 BC00462 V=500.0
'------------------------
'W62.5
'------------------------
MOVL C00463 BC00463 V=166.7 PL=0
REFP 3 C00464 BC00464
CALL JOB:SEARCH-R1
IMOV P0056 V=23.0 PL=0
SET P0351 P0006
SFTON P0351
REFP 3 C00465 BC00465
CALL JOB:SEARCH-R1
SET P0351 P0006
SFTON P0351
MOVL C00466 BC00466 V=250.0 PL=0
SFTOF
'PRZEJAZD
MOVL C00467 BC00467 V=500.0
MOVL C00468 BC00468 V=500.0
MOVL C00469 BC00469 V=500.0
MOVL C00470 BC00470 V=166.7 PL=0
REFP 3 C00471 BC00471
CALL JOB:SEARCH-R1
IMOV P0056 V=23.0 PL=0
SET P0352 P0006
SFTON P0352
REFP 3 C00472 BC00472
CALL JOB:SEARCH-R1
SET P0352 P0006
SFTON P0352
MOVL C00473 BC00473 V=250.0 PL=0
SFTOF
MOVL C00474 BC00474 V=500.0
'------------------------
'W29.8
'------------------------
MOVL C00475 BC00475 V=166.7 PL=0
REFP 3 C00476 BC00476
CALL JOB:SEARCH-R1
IMOV P0056 V=23.0 PL=0
SET P0353 P0006
SFTON P0353
REFP 3 C00477 BC00477
CALL JOB:SEARCH-R1
SET P0353 P0006
SFTON P0353
MOVL C00478 BC00478 V=250.0 PL=0
SFTOF
MOVL C00479 BC00479 V=500.0
'PRZEJAZD
MOVL C00480 BC00480 V=500.0
MOVJ C00481 BC00481 VJ=20.00
MOVJ C00482 BC00482 VJ=20.00
MOVL C00483 BC00483 V=500.0
MOVL C00484 BC00484 V=500.0
MOVL C00485 BC00485 V=500.0
'------------------------
'W29.11
'------------------------
MOVL C00486 BC00486 V=166.7 PL=0
REFP 3 C00487 BC00487
CALL JOB:SEARCH-R1
IMOV P0056 V=23.0 PL=0
SET P0354 P0006
SFTON P0354
REFP 3 C00488 BC00488
CALL JOB:SEARCH-R1
SET P0354 P0006
SFTON P0354
MOVL C00489 BC00489 V=250.0 PL=0
SFTOF
'PRZEJAZD
MOVL C00490 BC00490 V=500.0
'------------------------
'W29.14
'------------------------
MOVL C00491 BC00491 V=166.7 PL=0
REFP 3 C00492 BC00492
CALL JOB:SEARCH-R1
IMOV P0056 V=23.0 PL=0
SET P0355 P0006
SFTON P0355
REFP 3 C00493 BC00493
CALL JOB:SEARCH-R1
SET P0355 P0006
SFTON P0355
MOVL C00494 BC00494 V=250.0 PL=0
SFTOF
'PRZEJAZD
MOVL C00495 BC00495 V=500.0
'------------------------
'W63.17
'------------------------
MOVL C00496 BC00496 V=166.7 PL=0
REFP 3 C00497 BC00497
CALL JOB:SEARCH-R1
IMOV P0056 V=23.0 PL=0
SET P0356 P0006
SFTON P0356
REFP 3 C00498 BC00498
CALL JOB:SEARCH-R1
SET P0356 P0006
SFTON P0356
MOVL C00499 BC00499 V=250.0 PL=0
SFTOF
MOVL C00500 BC00500 V=500.0
MOVL C00501 BC00501 V=166.7 PL=0
REFP 3 C00502 BC00502
CALL JOB:SEARCH-R1
IMOV P0056 V=23.0 PL=0
SET P0357 P0006
SFTON P0357
REFP 3 C00503 BC00503
CALL JOB:SEARCH-R1
SET P0357 P0006
SFTON P0357
MOVL C00504 BC00504 V=250.0 PL=0
SFTOF
MOVL C00505 BC00505 V=500.0
MOVL C00506 BC00506 V=500.0
MOVL C00507 BC00507 V=416.7
MOVL C00508 BC00508 V=500.0
MOVL C00509 BC00509 V=166.7 PL=0
REFP 3 C00510 BC00510
CALL JOB:SEARCH-R1
IMOV P0056 V=23.0 PL=0
SET P0358 P0006
SFTON P0358
REFP 3 C00511 BC00511
CALL JOB:SEARCH-R1
SET P0358 P0006
SFTON P0358
MOVL C00512 BC00512 V=250.0 PL=0
SFTOF
MOVL C00513 BC00513 V=500.0
MOVL C00514 BC00514 V=166.7 PL=0
REFP 3 C00515 BC00515
CALL JOB:SEARCH-R1
IMOV P0056 V=23.0 PL=0
SET P0359 P0006
SFTON P0359
REFP 3 C00516 BC00516
CALL JOB:SEARCH-R1
SET P0359 P0006
SFTON P0359
MOVL C00517 BC00517 V=250.0 PL=0
SFTOF
COMM PAUSE
COMM 'PRZEJAZD
COMM MOVL C00518 BC00518 V=500.0
COMM MOVJ C00519 BC00519 VJ=30.00
COMM MOVJ C00520 BC00520 VJ=30.00
COMM MOVL C00521 BC00521 V=500.0
COMM MOVL C00522 BC00522 V=500.0
COMM '------------------------
COMM 'W62.20
COMM '------------------------
COMM MOVL C00523 BC00523 V=166.7 PL=0
COMM REFP 3 C00524 BC00524
COMM CALL JOB:SEARCH-R1
COMM IMOV P0056 V=23.0 PL=0
COMM SET P0358 P0006
COMM SFTON P0358
COMM REFP 3 C00525 BC00525
COMM CALL JOB:SEARCH-R1
COMM SET P0358 P0006
COMM SFTON P0358
COMM MOVL C00526 BC00526 V=250.0 PL=0
COMM SFTOF
COMM 'PRZEJAZD
COMM MOVL C00527 BC00527 V=500.0
COMM '------------------------
COMM 'W63.23
COMM '------------------------
COMM MOVL C00528 BC00528 V=166.7 PL=0
COMM REFP 3 C00529 BC00529
COMM CALL JOB:SEARCH-R1
COMM IMOV P0056 V=23.0 PL=0
COMM SET P0359 P0006
COMM SFTON P0359
COMM REFP 3 C00530 BC00530
COMM CALL JOB:SEARCH-R1
COMM SET P0359 P0006
COMM SFTON P0359
COMM MOVL C00531 BC00531 V=250.0 PL=0
COMM MOVL C00532 BC00532 V=500.0
COMM '------------------------
COMM 'W29.29
COMM '------------------------
COMM MOVL C00533 BC00533 V=166.7 PL=0
COMM REFP 3 C00534 BC00534
COMM CALL JOB:SEARCH-R1
COMM IMOV P0056 V=23.0 PL=0
COMM SET P0360 P0006
COMM SFTON P0360
COMM REFP 3 C00535 BC00535
COMM CALL JOB:SEARCH-R1
COMM SET P0360 P0006
COMM SFTON P0360
COMM MOVL C00536 BC00536 V=250.0 PL=0
COMM SFTOF
COMM 'PRZEJAZD
COMM MOVL C00537 BC00537 V=500.0
COMM MOVL C00538 BC00538 V=166.7 PL=0
COMM REFP 3 C00539 BC00539
COMM CALL JOB:SEARCH-R1
COMM IMOV P0056 V=23.0 PL=0
COMM SET P0361 P0006
COMM SFTON P0361
COMM REFP 3 C00540 BC00540
COMM CALL JOB:SEARCH-R1
COMM SET P0361 P0006
COMM SFTON P0361
COMM MOVL C00541 BC00541 V=250.0 PL=0
SFTOF
'------------------------
'W29.32
'------------------------
'PRZEJAZD
MOVL C00542 BC00542 V=500.0
MOVL C00543 BC00543 V=500.0
MOVL C00544 BC00544 V=416.7
MOVL C00545 BC00545 V=166.7 PL=0
REFP 3 C00546 BC00546
CALL JOB:SEARCH-R1
IMOV P0056 V=23.0 PL=0
SET P0362 P0006
SFTON P0362
REFP 3 C00547 BC00547
CALL JOB:SEARCH-R1
SET P0362 P0006
SFTON P0362
MOVL C00548 BC00548 V=250.0 PL=0
SFTOF
MOVJ C00549 BC00549 VJ=20.00
MOVJ C00550 BC00550 VJ=30.00
MOVJ C00551 BC00551 VJ=30.00
'KONIEC SEARCH WEW STRONA
MOVJ C00552 BC00552 VJ=30.00
MOVJ C00553 BC00553 VJ=20.00
MOVJ C00554 BC00554 VJ=10.00
MOVJ C00555 BC00555 VJ=20.00
MOVJ C00556 BC00556 VJ=20.00
'------------------------
'W29.2
'------------------------
MOVL C00557 BC00557 V=500.0
'------------------------
'W63.5
MACRO1 MJ#(0) ARGF9
'------------------------
SFTOF
SFTON P0301
MOVL C00558 BC00558 V=166.7 PL=0
ARCON
MOVL C00559 BC00559 V=8.3
ARCOF
SFTOF
MOVL C00560 BC00560 V=500.0
MACRO1 MJ#(0) ARGF24
SFTON P0302
MOVL C00561 BC00561 V=166.7 PL=0
ARCON
MOVL C00562 BC00562 V=8.3
ARCOF
MOVL C00563 BC00563 V=166.7 PL=0
SFTOF
MOVL C00564 BC00564 V=500.0
SFTON P0303
MOVL C00565 BC00565 V=166.7 PL=0
ARCON
MOVL C00566 BC00566 V=8.3
ARCOF
SFTOF
MOVL C00567 BC00567 V=166.7 PL=0
MOVL C00568 BC00568 V=500.0
MOVJ C00569 BC00569 VJ=30.00
MOVJ C00570 BC00570 VJ=20.00
MOVJ C00571 BC00571 VJ=30.00
MOVJ C00572 BC00572 VJ=30.00
MOVL C00573 BC00573 V=500.0
'------------------------
'W29.14
'------------------------
SFTON P0304
MOVL C00574 BC00574 V=166.7 PL=0
ARCON
MOVL C00575 BC00575 V=8.3
ARCOF
MOVL C00576 BC00576 V=166.7 PL=0
SFTOF
'PRZEJAZD
MOVL C00577 BC00577 V=500.0
MOVL C00578 BC00578 V=500.0
'------------------------
'W63.17
'------------------------
SFTON P0305
MOVL C00579 BC00579 V=166.7 PL=0
ARCON
MOVL C00580 BC00580 V=8.3
ARCOF
MOVL C00581 BC00581 V=166.7 PL=0
SFTOF
MOVL C00582 BC00582 V=500.0
SFTON P0306
MOVL C00583 BC00583 V=166.7
ARCON
MOVL C00584 BC00584 V=8.3
ARCOF
MOVL C00585 BC00585 V=166.7 PL=0
SFTOF
'PRZEJAZD
MOVL C00586 BC00586 V=500.0
SFTON P0307
MOVL C00587 BC00587 V=166.7
ARCON
MOVL C00588 BC00588 V=8.3
ARCOF
MOVL C00589 BC00589 V=166.7 PL=0
SFTOF
MOVL C00590 BC00590 V=500.0
MOVL C00591 BC00591 V=500.0
MOVL C00592 BC00592 V=333.3
MOVL C00593 BC00593 V=500.0
SFTON P0308
MOVL C00594 BC00594 V=166.7
ARCON
MOVL C00595 BC00595 V=8.3
ARCOF
MOVL C00596 BC00596 V=166.7 PL=0
SFTOF
MOVL C00597 BC00597 V=500.0
SFTON P0309
MOVL C00598 BC00598 V=166.7
ARCON
MOVL C00599 BC00599 V=8.3
ARCOF
MOVL C00600 BC00600 V=166.7 PL=0
SFTOF
COMM PAUSE
COMM MOVJ C00601 BC00601 VJ=20.00
COMM MOVJ C00602 BC00602 VJ=20.00
COMM MOVJ C00603 BC00603 VJ=30.00
COMM MOVJ C00604 BC00604 VJ=30.00
COMM MOVL C00605 BC00605 V=500.0
COMM '------------------------
COMM 'W63.20
COMM '------------------------
COMM SFTON P0308
COMM MOVL C00606 BC00606 V=166.7 PL=0
COMM ARCON
COMM MOVL C00607 BC00607 V=8.3
COMM ARCOF
COMM MOVL C00608 BC00608 V=166.7 PL=0
COMM SFTOF
COMM 'PRZEJAZD
COMM MOVL C00609 BC00609 V=500.0
COMM '------------------------
COMM 'W63.23
COMM '------------------------
COMM SFTON P0309
COMM MOVL C00610 BC00610 V=166.7 PL=0
COMM ARCON
COMM MOVL C00611 BC00611 V=8.3
COMM ARCOF
COMM MOVL C00612 BC00612 V=250.0 PL=0
COMM SFTOF
COMM MOVL C00613 BC00613 V=500.0
COMM SFTON P0310
COMM MOVL C00614 BC00614 V=166.7 PL=0
COMM ARCON
COMM MOVL C00615 BC00615 V=8.3
COMM ARCOF
COMM MOVL C00616 BC00616 V=250.0 PL=0
COMM SFTOF
COMM MOVL C00617 BC00617 V=500.0
COMM SFTON P0311
COMM MOVL C00618 BC00618 V=166.7 PL=0
COMM ARCON
COMM MOVL C00619 BC00619 V=8.3
COMM ARCOF
COMM MOVL C00620 BC00620 V=250.0 PL=0
SFTOF
MOVL C00621 BC00621 V=500.0
MOVL C00622 BC00622 V=500.0
MOVL C00623 BC00623 V=333.3
'------------------------
'W29.29
'------------------------
MOVL C00624 BC00624 V=500.0
SFTON P0312
COMM MOVL C00625 BC00625 V=166.7 PL=0
COMM ARCON
COMM MOVL C00626 BC00626 V=8.3
COMM ARCOF
COMM MOVL C00627 BC00627 V=250.0 PL=0
COMM MOVL C00628 BC00628 V=500.0
MOVL C00629 BC00629 V=166.7
ARCON
MOVL C00630 BC00630 V=8.3
ARCOF
SFTOF
'PRZEJAZD
MOVL C00631 BC00631 V=333.3
'PRZEJAZD
'KONIEC SPAWANIA CZESCI WSPOLNEJ
MOVJ C00632 BC00632 VJ=20.00
MOVJ C00633 BC00633 VJ=50.00
MOVJ C00634 BC00634 VJ=20.00
MOVJ C00635 BC00635 VJ=10.00
MOVJ C00636 BC00636 VJ=20.00
MOVJ C00637 BC00637 VJ=20.00
'------------------------
'W28.2
'------------------------
MOVJ C00638 BC00638 VJ=10.00
MOVJ C00639 BC00639 VJ=10.00
MOVL C00640 BC00640 V=500.0
MOVL C00641 BC00641 V=500.0
'------------------------
'W62.5
'------------------------
SFTON P0351
MOVL C00642 BC00642 V=166.7 PL=0
ARCON
MOVL C00643 BC00643 V=8.3
ARCOF
MOVL C00644 BC00644 V=250.0 PL=0
SFTOF
'PRZEJAZD
MOVL C00645 BC00645 V=500.0
MOVL C00646 BC00646 V=500.0
MOVL C00647 BC00647 V=500.0
SFTON P0352
MOVL C00648 BC00648 V=166.7 PL=0
ARCON
MOVL C00649 BC00649 V=8.3
ARCOF
MOVL C00650 BC00650 V=250.0 PL=0
SFTOF
MOVL C00651 BC00651 V=500.0
'------------------------
'W29.8
'------------------------
SFTON P0353
MOVL C00652 BC00652 V=166.7 PL=0
ARCON
MOVL C00653 BC00653 V=8.3
ARCOF
MOVL C00654 BC00654 V=250.0 PL=0
SFTOF
MOVL C00655 BC00655 V=500.0
'PRZEJAZD
MOVL C00656 BC00656 V=500.0
MOVJ C00657 BC00657 VJ=20.00
MOVL C00658 BC00658 V=500.0
MOVL C00659 BC00659 V=500.0
MOVL C00660 BC00660 V=500.0
'------------------------
'W29.11
'------------------------
SFTON P0354
MOVL C00661 BC00661 V=166.7 PL=0
ARCON
MOVL C00662 BC00662 V=8.3
ARCOF
MOVL C00663 BC00663 V=250.0 PL=0
SFTOF
'PRZEJAZD
MOVL C00664 BC00664 V=500.0
'------------------------
'W29.14
'------------------------
SFTON P0355
MOVL C00665 BC00665 V=166.7 PL=0
ARCON
MOVL C00666 BC00666 V=8.3
ARCOF
MOVL C00667 BC00667 V=250.0 PL=0
SFTOF
'PRZEJAZD
MOVL C00668 BC00668 V=500.0
'------------------------
'W63.17
'------------------------
SFTON P0356
MOVL C00669 BC00669 V=166.7 PL=0
ARCON
MOVL C00670 BC00670 V=8.3
ARCOF
MOVL C00671 BC00671 V=250.0 PL=0
SFTOF
MOVL C00672 BC00672 V=500.0
SFTON P0357
MOVL C00673 BC00673 V=166.7 PL=0
ARCON
MOVL C00674 BC00674 V=8.3
ARCOF
MOVL C00675 BC00675 V=250.0 PL=0
SFTOF
MOVL C00676 BC00676 V=500.0
MOVL C00677 BC00677 V=500.0
MOVL C00678 BC00678 V=416.7
MOVL C00679 BC00679 V=500.0
SFTON P0358
MOVL C00680 BC00680 V=166.7 PL=0
ARCON
MOVL C00681 BC00681 V=8.3
ARCOF
MOVL C00682 BC00682 V=250.0 PL=0
SFTOF
MOVL C00683 BC00683 V=500.0
SFTON P0359
MOVL C00684 BC00684 V=166.7 PL=0
ARCON
MOVL C00685 BC00685 V=8.3
ARCOF
MOVL C00686 BC00686 V=250.0 PL=0
SFTOF
COMM PAUSE
COMM PAUSE
COMM 'PRZEJAZD
COMM MOVL C00687 BC00687 V=500.0
COMM MOVJ C00688 BC00688 VJ=30.00
COMM MOVJ C00689 BC00689 VJ=30.00
COMM MOVJ C00690 BC00690 VJ=30.00
COMM MOVL C00691 BC00691 V=500.0
COMM MOVL C00692 BC00692 V=500.0
COMM '------------------------
COMM 'W62.20
COMM '------------------------
COMM SFTON P0358
COMM MOVL C00693 BC00693 V=166.7 PL=0
COMM ARCON
COMM MOVL C00694 BC00694 V=8.3
COMM ARCOF
COMM MOVL C00695 BC00695 V=250.0 PL=0
COMM SFTOF
COMM 'PRZEJAZD
COMM MOVL C00696 BC00696 V=500.0
COMM '------------------------
COMM 'W63.23
COMM '------------------------
COMM SFTON P0359
COMM MOVL C00697 BC00697 V=166.7 PL=0
COMM ARCON
COMM MOVL C00698 BC00698 V=8.3
COMM ARCOF
COMM MOVL C00699 BC00699 V=250.0 PL=0
COMM MOVL C00700 BC00700 V=500.0
COMM '------------------------
COMM 'W29.29
COMM '------------------------
COMM SFTON P0360
COMM MOVL C00701 BC00701 V=166.7 PL=0
COMM ARCON
COMM MOVL C00702 BC00702 V=8.3
COMM ARCOF
COMM MOVL C00703 BC00703 V=250.0 PL=0
COMM SFTOF
COMM 'PRZEJAZD
COMM MOVL C00704 BC00704 V=500.0
COMM SFTON P0361
COMM MOVL C00705 BC00705 V=166.7 PL=0
COMM ARCON
COMM MOVL C00706 BC00706 V=8.3
COMM ARCOF
COMM MOVL C00707 BC00707 V=250.0 PL=0
SFTOF
'------------------------
'W29.32
'------------------------
'PRZEJAZD
MOVL C00708 BC00708 V=500.0
MOVL C00709 BC00709 V=500.0
MOVL C00710 BC00710 V=416.7
MOVL C00711 BC00711 V=500.0
SFTON P0362
COMM MOVL C00712 BC00712 V=166.7 PL=0
COMM ARCON
COMM MOVL C00713 BC00713 V=8.3
COMM ARCOF
COMM MOVL C00714 BC00714 V=250.0 PL=0
COMM MOVL C00715 BC00715 V=500.0
MOVL C00716 BC00716 V=166.7
ARCON
MOVL C00717 BC00717 V=8.3
ARCOF
MOVL C00718 BC00718 V=250.0
SFTOF
MOVJ C00719 BC00719 VJ=20.00
MOVJ C00720 BC00720 VJ=30.00
MOVJ C00721 BC00721 VJ=30.00
MOVJ C00722 BC00722 VJ=30.00
CALL JOB:MOVE_OUT_OF_TUNNEL
END
